// TwinCAT 3 PLC project EngineeringToolbox
// Title: EngineeringToolbox
// Company: Beckhoff Electronics Mfg
// Author: Daniel Schlingmann
// ProjectVersion: 3.1.2.3
// Description: Engineering Toolbox Library The library is provided "as-is" for TwinCAT3.1 by the Beckhoff Industry Management for Electronics Manufacturing. Please check the function "DisclaimerStatement : WSTRING[1500]" in additon to the following disclaimer: THE SOFTWARE IS PROVIDED "AS IS", WITHOUT WARRANTY OF ANY KIND, EXPRESS OR IMPLIED, INCLUDING BUT NOT LIMITED TO THE WARRANTIES OF MERCHANTABILITY, FITNESS FOR A PARTICULAR PURPOSE AND NONINFRINGEMENT. IN NO EVENT SHALL THE AUTHORS OR COPYRIGHT HOLDERS BE LIABLE FOR ANY CLAIM, DAMAGES OR OTHER LIABILITY, WHETHER IN AN ACTION OF CONTRACT, TORT OR OTHERWISE, ARISING FROM, OUT OF OR IN CONNECTION WITH THE SOFTWARE OR THE USE OR OTHER DEALINGS IN THE SOFTWARE.
// ProgramVersion: 3.1.4022.7
// libraries:
//   Tc2_Drive, * (Beckhoff Automation GmbH)
//   Tc2_EtherCAT, * (Beckhoff Automation GmbH)
//   Tc2_IoFunctions, * (Beckhoff Automation GmbH)
//   Tc2_Math, * (Beckhoff Automation GmbH)
//   Tc2_MC2, * (Beckhoff Automation GmbH)
//   Tc2_MC2_Camming, * (Beckhoff Automation GmbH)
//   Tc2_MC2_Drive, * (Beckhoff Automation GmbH)
//   Tc2_MC2_FlyingSaw, * (Beckhoff Automation GmbH)
//   Tc2_MDP, * (Beckhoff Automation GmbH)
//   Tc2_ModbusRTU, * (Beckhoff Automation GmbH)
//   Tc2_ModbusSrv, * (Beckhoff Automation GmbH)
//   Tc2_NC, * (Beckhoff Automation GmbH)
//   Tc2_NCI, * (Beckhoff Automation GmbH)
//   Tc2_NcKinematicTransformation, * (Beckhoff Automation GmbH)
//   Tc2_PlcInterpolation, * (Beckhoff Automation GmbH)
//   Tc2_SerialCom, * (Beckhoff Automation GmbH)
//   Tc2_Smtp, * (Beckhoff Automation GmbH)
//   Tc2_Standard, * (Beckhoff Automation GmbH)
//   Tc2_SUPS, * (Beckhoff Automation GmbH)
//   Tc2_System, * (Beckhoff Automation GmbH)
//   Tc2_TcpIp, * (Beckhoff Automation GmbH)
//   Tc2_Utilities, * (Beckhoff Automation GmbH)
//   Tc2_XmlDataSrv, * (Beckhoff Automation GmbH)
//   Tc3_Module, * (Beckhoff Automation GmbH)
//   Tc2_BackupRestoreEL6900,newest,Beckhoff Automation GmbH
// project tree:
//   GVLs/ Gvl.TcGVL, PARAM.TcGVL
//   POUs/BoundsCheck/ boundsError.TcPOU (not stored), boundsOK.TcPOU (not stored), checkBounds.TcPOU, CheckBoundsInfo.TcPOU
//   POUs/Connectivity/ADS/ AdsDataExchange.TcPOU (not stored)
//   POUs/Connectivity/ Ipv4Addr_TO_UDINT.TcPOU (not stored), U_DEVICE_COM_CACHE.TcDUT (not stored), U_IPv4Addr.TcDUT (not stored), isValidIPv4Addr.TcPOU
//   POUs/Connectivity/TF6310-TcpServer/DeviceCom/ TCPDeviceCom_SendRecBytes.TcPOU (not stored), TCPDeviceCom_SendRecString.TcPOU
//   POUs/Connectivity/TF6340-SerialCom/ComPortDeviceCom/ ComPortDeviceCom_BufferHandle.TcPOU, ComPortDeviceCom_SendRecBytes.TcPOU, ComPortDeviceCom_SendRecString.TcPOU (not stored), ComPortEL6x22BEasyConnect.TcPOU (not stored)
//   POUs/Connectivity/TF6340-SerialCom/ComPortBasic/ ComPortBackground.TcPOU (not stored), ComPortSendRec.TcPOU
//   POUs/Connectivity/TF625x-Modbus/Master/TF6250-ModbusTcpServer/TCP/ ModbusTcpMaster.TcPOU
//   POUs/Connectivity/TF625x-Modbus/Master/TF6250-ModbusTcpServer/UDP/ ModbusUdpMaster.TcPOU
//   POUs/Connectivity/TF625x-Modbus/Master/TF6255-ModbusRtu/ ModbusRtuMaster22B.TcPOU, ModbusRtuMaster5B.TcPOU (not stored), ModbusRtuMasterPC.TcPOU
//   POUs/Connectivity/TF625x-Modbus/Master/_Components/ ModbusJob.TcPOU (not stored), ModbusSlaveCom.TcPOU
//   POUs/Connectivity/TF625x-Modbus/Slave/ ModbusSlaveBase.TcPOU (not stored)
//   POUs/Connectivity/TF6310-TcpServer/TcpBasic/ TCPSendRecCtrl.TcPOU (not stored), TCPConnectionCtrl.TcPOU, TCPSocketCtrl.TcPOU (not stored)
//   POUs/Connectivity/TF6310-TcpServer/UdpBasic/ UDPSendRecCtrl.TcPOU (not stored), UDPServerCtrl.TcPOU (not stored), UDPSocketCtrl.TcPOU (not stored)
//   POUs/ControllerTools/ AverageFilter.TcPOU (not stored), PIDController.TcPOU (not stored), PT1Filter.TcPOU (not stored), signum.TcPOU (not stored), SlewRateLimitter.TcPOU, SlidingAverageExt.TcPOU, SlidingAverage.TcPOU, ThreePointController.TcPOU
//   POUs/DataBuffer/ DoubleBuffer.TcPOU (not stored), Quicksort.TcPOU (not stored)
//   POUs/DataBuffer/Fifo/ Fifo.TcPOU (not stored), FifoExt.TcPOU, FifoLRealSimple.TcPOU, FifoBase.TcPOU
//   POUs/DataBuffer/Ringbuffer/ RingbufferBase.TcPOU, Ringbuffer.TcPOU (not stored), RingbufferCharSimple.TcPOU (not stored), RingbufferExt.TcPOU (not stored), RingbufferByteSimple.TcPOU (not stored), RingbufferLRealSimple.TcPOU
//   POUs/EventLogger/ EventsWriteToLogbook.TcPOU (not stored), EVENT_HANDLING_CONFIG.TcDUT (not stored), getEventClassPriority.TcPOU (not stored), getEventClassText.TcPOU (not stored), SOURCE_ID.TcDUT (not stored)
//   POUs/EventLogger/ReadEvents/ EventlogRead.TcPOU (not stored), EVENTLOG_READ_DATA.TcDUT (not stored), EVENTLOG_READ_HANDLEINFO.TcDUT (not stored), EVENTLOG_READ_STREAM.TcDUT (not stored), EVENTLOG_READ_STREAM_DATA_RAW.TcDUT (not stored), EVENTLOG_READ_STREAM_DATA_RAW_EX.TcDUT
//   POUs/EventLogger/TriggerEvents/ EventHandling.TcPOU, EventHandlingGrp10.TcPOU (not stored), EventHandlingGrp25.TcPOU, EventHandlingGrp50.TcPOU (not stored), EventHandlingGrpCustomized.TcPOU (not stored), EventHandlingConfirmIsReq.TcPOU (not stored), EventHandlingStatisticInfo.TcPOU
//   POUs/Fieldbus/CANopen/ CANopenMasterDiag.TcPOU (not stored), CANopenMasterIO.TcPOU
//   POUs/Fieldbus/EAP/ EAP_PUB_SUB_IO.TcPOU (not stored), EAP_DEVICE_IO.TcPOU (not stored), EAP_PUB_VAR.TcPOU, EAP_SUB_VAR.TcPOU (not stored)
//   POUs/Fieldbus/EtherCAT/ EcCoEReadNewestDiagMsg.TcPOU, EcDiagBase.TcPOU, EcDiagBase_wEvents.TcPOU
//   POUs/Fieldbus/EtherCAT/_Components/ EcMasterIO.TcPOU (not stored), EcMasterSupervisor.TcPOU (not stored), EcSlavesDiag.TcPOU (not stored), EcSlaveSupervisor.TcPOU, EC_MASTER_DEVICE_STATE.TcDUT, EC_SLAVE_DIAG_INFO_DATA.TcDUT (not stored)
//   POUs/Fieldbus/Profibus/ ProfibusMasterDiag.TcPOU (not stored), ProfibusMasterIO.TcPOU (not stored)
//   POUs/Fieldbus/Profinet/ ProfinetControllerIO.TcPOU (not stored), ProfinetControllerIO_wEvents.TcPOU (not stored), ProfinetDeviceIO.TcPOU (not stored)
//   POUs/FileHandling/Basic/ FileHandling.TcPOU, ReadDirSimple.TcPOU (not stored), ReadDirSimpleExt.TcPOU
//   POUs/FileHandling/TF6421-XmlServer/ XmlReadWrite.TcPOU (not stored), XmlReadWriteWithBackupFile.TcPOU (not stored)
//   POUs/IO/Analog/ AnalogIn.TcPOU, AnalogIn32.TcPOU, AnalogInELMBase.TcPOU (not stored), AnalogInELMSingleSampleDINT.TcPOU, AnalogInELMSingleSampleREAL.TcPOU (not stored), AnalogInREAL.TcPOU, AnalogOut.TcPOU (not stored)
//   POUs/IO/ BlowOffSensors.TcPOU (not stored), Button.TcPOU, ButtonExt.TcPOU (not stored), Fuse.TcPOU (not stored), InOut.TcPOU (not stored), InOutExt.TcPOU (not stored), Input.TcPOU (not stored), Output.TcPOU (not stored)
//   POUs/IO/Cylinder/ Cylinder.TcPOU, CylinderExt.TcPOU (not stored), CylinderType4.TcPOU, I_Cylinder.TcIO (not stored)
//   POUs/IO/Drives/ AxDriveBase.TcPOU (not stored), AxDriveGetRef.TcPOU (not stored), I_AxDriveBase.TcIO
//   POUs/IO/Drives/CoE/ AxDriveCoE.TcPOU, AxDriveCoE_wEvents.TcPOU, CiA_DS402Controlword.TcPOU (not stored), CiA_DS402Statusword.TcPOU (not stored), eCiA_DS402_CONTROL_CMD.TcDUT, eCiA_DS402_STATUS_STATE.TcDUT (not stored)
//   POUs/IO/Drives/CoE/EL72xx/ AxDriveCoE_EL72xxParam.TcPOU (not stored), CiA_DS402StatuswordEx7xxx.TcPOU
//   POUs/IO/Drives/DC/Ey73xx/ AxDriveDC.TcPOU (not stored), AxDriveDC_wEvents.TcPOU (not stored)
//   POUs/IO/Drives/SoE/ AxDriveSoE_Ax5000CommutationCalib.TcPOU (not stored), AxDriveSoE_Ax5000CalcPower.TcPOU (not stored), AxDriveSoE_Ax5000SwitchParamSet.TcPOU (not stored), Ax580x.TcPOU (not stored), AxDriveSoE_Ax5000.TcPOU, AxDriveSoE_Ax5000Param.TcPOU, AxDriveSoE_Ax5000wEvents.TcPOU, AxDriveSoE_Rexroth.TcPOU (not stored)
//   POUs/IO/Drives/SoE/Ax5000ParamSTRUCTs/P/ AX5000_P_0001.TcDUT (not stored), AX5000_P_0002.TcDUT (not stored), AX5000_P_0003.TcDUT (not stored), AX5000_P_0004.TcDUT (not stored), AX5000_P_0009.TcDUT, AX5000_P_0010.TcDUT, AX5000_P_0020.TcDUT, AX5000_P_0021.TcDUT (not stored), AX5000_P_0040.TcDUT (not stored), AX5000_P_0050.TcDUT, AX5000_P_0051.TcDUT, AX5000_P_0052.TcDUT (not stored), AX5000_P_0053.TcDUT, AX5000_P_0054.TcDUT (not stored), AX5000_P_0055.TcDUT (not stored), AX5000_P_0056.TcDUT, AX5000_P_0057.TcDUT, AX5000_P_0058.TcDUT (not stored), AX5000_P_0059.TcDUT, AX5000_P_0060.TcDUT (not stored), AX5000_P_0061.TcDUT, AX5000_P_0062.TcDUT (not stored), AX5000_P_0063.TcDUT (not stored), AX5000_P_0064.TcDUT (not stored), AX5000_P_0065.TcDUT, AX5000_P_0066.TcDUT (not stored), AX5000_P_0067.TcDUT, AX5000_P_0068.TcDUT (not stored), AX5000_P_0069.TcDUT (not stored), AX5000_P_0070.TcDUT, AX5000_P_0071.TcDUT (not stored), AX5000_P_0072.TcDUT (not stored), AX5000_P_0073.TcDUT (not stored), AX5000_P_0074.TcDUT (not stored), AX5000_P_0075.TcDUT (not stored), AX5000_P_0076.TcDUT (not stored), AX5000_P_0077.TcDUT (not stored), AX5000_P_0078.TcDUT, AX5000_P_0088.TcDUT, AX5000_P_0089.TcDUT (not stored), AX5000_P_0090.TcDUT (not stored), AX5000_P_0091.TcDUT (not stored), AX5000_P_0092.TcDUT (not stored), AX5000_P_0093.TcDUT, AX5000_P_0096.TcDUT (not stored), AX5000_P_0097.TcDUT, AX5000_P_0098_beckhoff.TcDUT (not stored), AX5000_P_0098_beckhoff_electrical_data.TcDUT (not stored), AX5000_P_0099.TcDUT (not stored), AX5000_P_0100.TcDUT (not stored), AX5000_P_0101.TcDUT (not stored), AX5000_P_0102.TcDUT (not stored), AX5000_P_0103.TcDUT (not stored), AX5000_P_0104.TcDUT (not stored), AX5000_P_0105.TcDUT (not stored), AX5000_P_0106.TcDUT (not stored), AX5000_P_0107.TcDUT (not stored), AX5000_P_0108.TcDUT (not stored), AX5000_P_0109.TcDUT (not stored), AX5000_P_0110.TcDUT, AX5000_P_0111.TcDUT (not stored), AX5000_P_0112.TcDUT (not stored), AX5000_P_0113.TcDUT (not stored), AX5000_P_0114.TcDUT, AX5000_P_0115.TcDUT (not stored), AX5000_P_0116.TcDUT (not stored), AX5000_P_0117.TcDUT (not stored), AX5000_P_0118.TcDUT (not stored), AX5000_P_0119.TcDUT, AX5000_P_0125.TcDUT (not stored), AX5000_P_0126.TcDUT (not stored), AX5000_P_0127.TcDUT (not stored), AX5000_P_0128.TcDUT (not stored), AX5000_P_0150.TcDUT (not stored), AX5000_P_0151.TcDUT (not stored), AX5000_P_0152.TcDUT, AX5000_P_0153.TcDUT (not stored), AX5000_P_0154.TcDUT, AX5000_P_0155.TcDUT (not stored), AX5000_P_0158.TcDUT, AX5000_P_0159.TcDUT, AX5000_P_0160.TcDUT (not stored), AX5000_P_0161.TcDUT (not stored), AX5000_P_0162.TcDUT, AX5000_P_0163.TcDUT (not stored), AX5000_P_0165.TcDUT (not stored), AX5000_P_0166.TcDUT, AX5000_P_0167.TcDUT (not stored), AX5000_P_0168.TcDUT (not stored), AX5000_P_0169.TcDUT, AX5000_P_0170.TcDUT (not stored), AX5000_P_0171.TcDUT (not stored), AX5000_P_0180.TcDUT (not stored), AX5000_P_0181.TcDUT (not stored), AX5000_P_0182.TcDUT (not stored), AX5000_P_0183.TcDUT (not stored), AX5000_P_0184.TcDUT (not stored), AX5000_P_0185.TcDUT (not stored), AX5000_P_0188.TcDUT, AX5000_P_0189.TcDUT (not stored), AX5000_P_0192.TcDUT (not stored), AX5000_P_0193.TcDUT (not stored), AX5000_P_0196.TcDUT, AX5000_P_0198.TcDUT (not stored), AX5000_P_0199.TcDUT (not stored), AX5000_P_0200.TcDUT (not stored), AX5000_P_0201.TcDUT (not stored), AX5000_P_0202.TcDUT (not stored), AX5000_P_0203.TcDUT (not stored), AX5000_P_0204.TcDUT (not stored), AX5000_P_0205.TcDUT, AX5000_P_0206.TcDUT (not stored), AX5000_P_0207.TcDUT, AX5000_P_0208.TcDUT, AX5000_P_0209.TcDUT (not stored), AX5000_P_0210.TcDUT (not stored), AX5000_P_0211.TcDUT (not stored), AX5000_P_0212.TcDUT, AX5000_P_0213.TcDUT, AX5000_P_0214.TcDUT (not stored), AX5000_P_0215.TcDUT, AX5000_P_0216.TcDUT (not stored), AX5000_P_0217.TcDUT (not stored), AX5000_P_0218.TcDUT (not stored), AX5000_P_0219.TcDUT, AX5000_P_0220.TcDUT (not stored), AX5000_P_0221.TcDUT (not stored), AX5000_P_0250.TcDUT (not stored), AX5000_P_0251.TcDUT, AX5000_P_0252.TcDUT, AX5000_P_0253.TcDUT, AX5000_P_0254.TcDUT (not stored), AX5000_P_0255.TcDUT, AX5000_P_0256.TcDUT, AX5000_P_0270.TcDUT (not stored), AX5000_P_0271.TcDUT (not stored), AX5000_P_0272.TcDUT (not stored), AX5000_P_0273.TcDUT, AX5000_P_0274.TcDUT (not stored), AX5000_P_0275.TcDUT, AX5000_P_0276.TcDUT (not stored), AX5000_P_0277.TcDUT (not stored), AX5000_P_0278.TcDUT (not stored), AX5000_P_0300.TcDUT (not stored), AX5000_P_0301.TcDUT, AX5000_P_0302.TcDUT (not stored), AX5000_P_0303.TcDUT (not stored), AX5000_P_0304.TcDUT, AX5000_P_0305.TcDUT (not stored), AX5000_P_0306.TcDUT (not stored), AX5000_P_0307.TcDUT (not stored), AX5000_P_0308.TcDUT, AX5000_P_0309.TcDUT (not stored), AX5000_P_0310.TcDUT, AX5000_P_0311.TcDUT (not stored), AX5000_P_0312.TcDUT, AX5000_P_0313.TcDUT (not stored), AX5000_P_0314.TcDUT, AX5000_P_0315.TcDUT, AX5000_P_0316.TcDUT, AX5000_P_0317.TcDUT (not stored), AX5000_P_0320.TcDUT (not stored), AX5000_P_0321.TcDUT (not stored), AX5000_P_0322.TcDUT (not stored), AX5000_P_0323.TcDUT, AX5000_P_0324.TcDUT (not stored), AX5000_P_0325.TcDUT (not stored), AX5000_P_0326.TcDUT (not stored), AX5000_P_0350.TcDUT, AX5000_P_0351.TcDUT (not stored), AX5000_P_0352.TcDUT (not stored), AX5000_P_0353.TcDUT (not stored), AX5000_P_0354.TcDUT (not stored), AX5000_P_0356.TcDUT, AX5000_P_0360.TcDUT, AX5000_P_0361.TcDUT (not stored), AX5000_P_0400.TcDUT (not stored), AX5000_P_0401.TcDUT (not stored), AX5000_P_0402.TcDUT, AX5000_P_0451.TcDUT, AX5000_P_0452.TcDUT (not stored), AX5000_P_0453.TcDUT (not stored), AX5000_P_0454.TcDUT (not stored), AX5000_P_0455.TcDUT (not stored), AX5000_P_0456.TcDUT (not stored), AX5000_P_0457.TcDUT, AX5000_P_0458.TcDUT (not stored), AX5000_P_0459.TcDUT, AX5000_P_0460.TcDUT (not stored), AX5000_P_0461.TcDUT, AX5000_P_0462.TcDUT (not stored), AX5000_P_0463.TcDUT (not stored), AX5000_P_0464.TcDUT (not stored), AX5000_P_0502.TcDUT (not stored), AX5000_P_0503.TcDUT (not stored), AX5000_P_0504.TcDUT, AX5000_P_0505.TcDUT (not stored), AX5000_P_0511.TcDUT, AX5000_P_0512.TcDUT (not stored), AX5000_P_0513.TcDUT (not stored), AX5000_P_0514.TcDUT (not stored), AX5000_P_0515.TcDUT, AX5000_P_0516.TcDUT (not stored), AX5000_P_0517.TcDUT, AX5000_P_0518.TcDUT, AX5000_P_0552.TcDUT (not stored), AX5000_P_0553.TcDUT, AX5000_P_0554.TcDUT, AX5000_P_0555.TcDUT (not stored), AX5000_P_0556.TcDUT (not stored), AX5000_P_0557.TcDUT (not stored), AX5000_P_0558.TcDUT (not stored), AX5000_P_0601.TcDUT, AX5000_P_0602.TcDUT (not stored), AX5000_P_0610.TcDUT (not stored), AX5000_P_0611.TcDUT (not stored), AX5000_P_0800.TcDUT (not stored), AX5000_P_0801.TcDUT, AX5000_P_0802.TcDUT (not stored), AX5000_P_0804.TcDUT (not stored), AX5000_P_0805.TcDUT (not stored), AX5000_P_0806.TcDUT, AX5000_P_0810.TcDUT (not stored), AX5000_P_0811.TcDUT (not stored), AX5000_P_0850.TcDUT, AX5000_P_0851.TcDUT, AX5000_P_0900.TcDUT (not stored), AX5000_P_0901.TcDUT (not stored), AX5000_P_0902.TcDUT, AX5000_P_0904.TcDUT (not stored), AX5000_P_0905.TcDUT (not stored), AX5000_P_0906.TcDUT (not stored), AX5000_P_0912.TcDUT, AX5000_P_1000.TcDUT (not stored), AX5000_P_1001.TcDUT, AX5000_P_1002.TcDUT (not stored), AX5000_P_1003.TcDUT (not stored), AX5000_P_1004.TcDUT (not stored), AX5000_P_1005.TcDUT (not stored), AX5000_P_1006.TcDUT (not stored), AX5000_P_1007.TcDUT, AX5000_P_1008.TcDUT, AX5000_P_1009.TcDUT (not stored), AX5000_P_1010.TcDUT (not stored), AX5000_P_1011.TcDUT (not stored), AX5000_P_1012.TcDUT (not stored), AX5000_P_1020.TcDUT (not stored), AX5000_P_1021.TcDUT (not stored), AX5000_P_1022.TcDUT, AX5000_P_2000.TcDUT, AX5000_P_2001.TcDUT, AX5000_P_2002.TcDUT
//   POUs/IO/Drives/SoE/Ax5000ParamSTRUCTs/S/ AX5000_S_0001.TcDUT, AX5000_S_0002.TcDUT (not stored), AX5000_S_0007.TcDUT (not stored), AX5000_S_0011.TcDUT, AX5000_S_0012.TcDUT (not stored), AX5000_S_0013.TcDUT, AX5000_S_0015.TcDUT, AX5000_S_0016.TcDUT (not stored), AX5000_S_0017.TcDUT (not stored), AX5000_S_0018.TcDUT, AX5000_S_0024.TcDUT (not stored), AX5000_S_0029.TcDUT (not stored), AX5000_S_0030.TcDUT, AX5000_S_0031.TcDUT, AX5000_S_0032.TcDUT (not stored), AX5000_S_0033.TcDUT (not stored), AX5000_S_0034.TcDUT (not stored), AX5000_S_0035.TcDUT (not stored), AX5000_S_0036.TcDUT (not stored), AX5000_S_0037.TcDUT, AX5000_S_0040.TcDUT (not stored), AX5000_S_0043.TcDUT (not stored), AX5000_S_0044.TcDUT (not stored), AX5000_S_0045.TcDUT (not stored), AX5000_S_0046.TcDUT (not stored), AX5000_S_0047.TcDUT (not stored), AX5000_S_0048.TcDUT, AX5000_S_0051.TcDUT (not stored), AX5000_S_0053.TcDUT, AX5000_S_0055.TcDUT (not stored), AX5000_S_0076.TcDUT (not stored), AX5000_S_0079.TcDUT (not stored), AX5000_S_0080.TcDUT, AX5000_S_0081.TcDUT, AX5000_S_0082.TcDUT (not stored), AX5000_S_0083.TcDUT (not stored), AX5000_S_0084.TcDUT (not stored), AX5000_S_0085.TcDUT (not stored), AX5000_S_0086.TcDUT, AX5000_S_0091.TcDUT, AX5000_S_0092.TcDUT (not stored), AX5000_S_0095.TcDUT, AX5000_S_0099.TcDUT, AX5000_S_0100.TcDUT, AX5000_S_0101.TcDUT (not stored), AX5000_S_0103.TcDUT (not stored), AX5000_S_0104.TcDUT, AX5000_S_0106.TcDUT, AX5000_S_0107.TcDUT (not stored), AX5000_S_0109.TcDUT (not stored), AX5000_S_0110.TcDUT (not stored), AX5000_S_0111.TcDUT, AX5000_S_0112.TcDUT (not stored), AX5000_S_0113.TcDUT (not stored), AX5000_S_0119.TcDUT, AX5000_S_0120.TcDUT (not stored), AX5000_S_0124.TcDUT (not stored), AX5000_S_0126.TcDUT, AX5000_S_0130.TcDUT (not stored), AX5000_S_0131.TcDUT, AX5000_S_0134.TcDUT, AX5000_S_0135.TcDUT (not stored), AX5000_S_0136.TcDUT (not stored), AX5000_S_0137.TcDUT (not stored), AX5000_S_0143.TcDUT (not stored), AX5000_S_0149.TcDUT (not stored), AX5000_S_0159.TcDUT, AX5000_S_0160.TcDUT, AX5000_S_0161.TcDUT, AX5000_S_0162.TcDUT, AX5000_S_0163.TcDUT, AX5000_S_0169.TcDUT (not stored), AX5000_S_0170.TcDUT (not stored), AX5000_S_0179.TcDUT, AX5000_S_0185.TcDUT, AX5000_S_0186.TcDUT (not stored), AX5000_S_0187.TcDUT, AX5000_S_0188.TcDUT, AX5000_S_0189.TcDUT (not stored), AX5000_S_0196.TcDUT (not stored), AX5000_S_0200.TcDUT, AX5000_S_0201.TcDUT (not stored), AX5000_S_0203.TcDUT (not stored), AX5000_S_0204.TcDUT (not stored), AX5000_S_0206.TcDUT (not stored), AX5000_S_0207.TcDUT (not stored), AX5000_S_0216.TcDUT, AX5000_S_0217.TcDUT, AX5000_S_0219.TcDUT (not stored), AX5000_S_0254.TcDUT (not stored), AX5000_S_0256.TcDUT (not stored), AX5000_S_0257.TcDUT (not stored), AX5000_S_0267.TcDUT, AX5000_S_0273.TcDUT (not stored), AX5000_S_0274.TcDUT, AX5000_S_0292.TcDUT (not stored), AX5000_S_0295.TcDUT (not stored), AX5000_S_0296.TcDUT (not stored), AX5000_S_0347.TcDUT (not stored), AX5000_S_0348.TcDUT (not stored), AX5000_S_0372.TcDUT, AX5000_S_0374.TcDUT (not stored), AX5000_S_0375.TcDUT, AX5000_S_0380.TcDUT, AX5000_S_0381.TcDUT (not stored), AX5000_S_0383.TcDUT, AX5000_S_0384.TcDUT (not stored), AX5000_S_0390.TcDUT (not stored), AX5000_S_0403.TcDUT (not stored), AX5000_S_0405.TcDUT (not stored), AX5000_S_0409.TcDUT (not stored), AX5000_S_0410.TcDUT (not stored), AX5000_S_0429.TcDUT, AX5000_S_0432.TcDUT (not stored), AX5000_S_0435.TcDUT, AX5000_S_0436.TcDUT (not stored)
//   POUs/IO/Drives/Stepper/ AxDriveStepper.TcPOU, AxDriveStepperParam.TcPOU (not stored), AxDriveStepper_wEvents.TcPOU (not stored)
//   POUs/IO/EL-EP/ AnalogOut_EL2535.TcPOU (not stored), EL1262_Base.TcPOU (not stored), EL3681.TcPOU (not stored), EL1904.TcPOU (not stored), EL69xx.TcPOU, EL3356.TcPOU (not stored), Eyx9xx.TcPOU, ZB8610.TcPOU
//   POUs/IO/EL-EP/EL9x/ EL9501.TcPOU (not stored), EL9576.TcPOU (not stored), EL95xxPowerTerminal.TcPOU, ELSystemTerminal.TcPOU
//   POUs/IO/_EcSlaveFWUpdater/ EcSlaveDevFWUpdater.TcPOU (not stored)
//   POUs/IO/_EcSlaveInfoDataIO/ EcSlaveInfoData.TcPOU (not stored), EcSlaveInfoDataExt.TcPOU (not stored), I_EcSlaveInfoData.TcIO
//   POUs/IO/EL-EP/EL3403/ EL3403.TcPOU (not stored), EL3403Logic.TcPOU
//   POUs/IO/EL-EP/EP92xxPwrBox/ EP9214.TcPOU, EP9214_CHANNEL.TcPOU (not stored), EP9224_0037.TcPOU, EP9224_0037_CHANNEL.TcPOU
//   POUs/IO/FreqConv/EtherCAT/DS402/ EcFcDS402_ComBase.TcPOU (not stored)
//   POUs/IO/FreqConv/ IOFcCom.TcPOU
//   POUs/IO/Motors/ IOMotor.TcPOU (not stored), IOMotor2Dir.TcPOU (not stored), IOMotorStarDelta.TcPOU (not stored)
//   POUs/IO/[underDev]/ Cylinder_wUnitItf.TcPOU
//   POUs/IO/_ItfActuators/ I_ActuatorBase.TcIO (not stored), I_ActuatorEnableDisable.TcIO (not stored), I_ActuatorFwdRev.TcIO, I_ActuatorFwdBwd.TcIO, I_ActuatorLeftRight.TcIO, I_ActuatorOnOff.TcIO (not stored), I_ActuatorOpenClose.TcIO (not stored), I_ActuatorPosNeg.TcIO (not stored), I_ActuatorStartStop.TcIO (not stored), I_ActuatorUpDown.TcIO (not stored), I_ActuatorWorkBase.TcIO (not stored)
//   POUs/IpcDiag/MDP/InfoModuls/ MDP_CPU.TcPOU, MDP_Fan.TcPOU, MDP_Mainboard.TcPOU (not stored), MDP_RaidSimple.TcPOU (not stored), MDP_ReadModulList.TcPOU (not stored), MDP_SiliconDrives.TcPOU, MDP_UPS.TcPOU (not stored)
//   POUs/IpcDiag/MDP/ MDP_Info.TcPOU, MDP_IpcDiag.TcPOU (not stored), MDP_IpcDiag_wEvents.TcPOU (not stored)
//   POUs/IpcDiag/ UPSStatus.TcPOU (not stored)
//   POUs/Logging/ DataFileLogger.TcPOU, DataUdpLogger.TcPOU (not stored), I_LogbookSubscriber.TcIO (not stored), I_Logbook.TcIO (not stored), Logbook.TcPOU (not stored), LogbookData.TcDUT, LogbookPuplisher.TcPOU, LogbookSubEventLog.TcPOU (not stored), LogbookSubSendMail.TcPOU, adsLogError.TcPOU, adsLogHint.TcPOU (not stored), adsLogWarn.TcPOU, LogbookSubSysLog.TcPOU, LogbookSubWriteFile.TcPOU, Logbook_wEventClass.TcPOU, adsLogwTcEventClass.TcPOU (not stored)
//   POUs/Motion/TF50xx-NC/00_Base/ I_AxNcPTP.TcIO (not stored), AxFbBase.TcPOU, AxRWParaBase.TcPOU (not stored), I_AxNcBase.TcIO
//   POUs/Motion/TF50xx-NC/02_Options/Parameter/ AxPara.TcPOU (not stored), AxParaCtrl.TcPOU
//   POUs/Motion/TF50xx-NC/03_Utilities/ AxAutoWriteSoftLimit.TcPOU, CoordinateTransformation2D.TcPOU (not stored), AxCalcPosBias.TcPOU, AxResonanceAvoidance.TcPOU (excluded from build), AxSoftSyncDistance.TcPOU (not stored), AxStatemodel.TcPOU (not stored), AxAutoFct.TcPOU (not stored), AX_JOB.TcPOU (not stored), getOvrVelo.TcPOU
//   POUs/Motion/TF50xx-NC/ AxNcPTPwJobs.TcPOU (not stored), AxNcBaseExt.TcPOU (not stored), AxNcPtpGear.TcPOU, AxNcBase.TcPOU, AxNcPTP.TcPOU (not stored)
//   POUs/Motion/TF5100-NCI/ NciChannel_wEvents.TcPOU (not stored), NciChannel.TcPOU (not stored)
//   POUs/Motion/TF511x-KIN/03_DUTs/Positions/ KIN_POSITIONS.TcPOU (not stored), KIN_POSITIONS_ACS_DUT.TcDUT (not stored), KIN_POSITIONS_MCS_DUT.TcDUT, U_KIN_POSITIONS.TcDUT
//   POUs/Motion/TF511x-KIN/03_DUTs/Trafo/ KIN_CALCTRAFO_AXPOS_PARAM.TcPOU (not stored), KIN_STATE_OBSERVER_OID_PARAM.TcPOU (not stored), KIN_STATICTRAFO_PARAM.TcPOU (not stored), KIN_TOOLTRAFO_PARAM.TcPOU, UCS.TcPOU (not stored)
//   POUs/Motion/ VALUE_3D.TcPOU (not stored), VALUE_3D_DUT.TcDUT (not stored), VALUE_6D.TcPOU (not stored), VALUE_6D_DUT.TcDUT
//   POUs/Safety/Diag/ SafetyLogicAndIOTerminalDiag.TcPOU (not stored), SafetyIODeviceDiagRead.TcPOU (not stored), SafetyIODeviceDiag_wEvents.TcPOU, SafetyIOsDiag.TcPOU, SafetyLogicTerminalDiag.TcPOU, SafetyPlcTerminalDiag.TcPOU
//   POUs/StringHelper/ CHR_TO_STR.TcPOU, cutStrNumberToSeperator.TcPOU (not stored), cutStrToSeperator2.TcPOU, replaceUmlauts.TcPOU, stringCmp.TcPOU, STR_TO_ASC.TcPOU (not stored), cutStrToSeperator.TcPOU (not stored), cutWStrToSeperator.TcPOU (not stored), DWORD_TO_BINSTR_EXT.TcPOU (not stored), DWORD_TO_HEXSTR_EXT.TcPOU (not stored), getCntCharInStr.TcPOU (not stored), getCntCharInWStr.TcPOU, isWStringNumeric.TcPOU (not stored), HEXSTR_TO_DWORD.TcPOU, HEXSTR_TO_LWORD.TcPOU, INSERT_EXT.TcPOU, LWORD_TO_BINSTR_EXT.TcPOU, LWORD_TO_HEXSTR_EXT.TcPOU, readStrToSeperator.TcPOU, replaceInString.TcPOU (not stored), getFilledString.TcPOU (not stored), isStringNumeric.TcPOU (not stored), readWStrToSeperator.TcPOU (not stored), replaceInWString.TcPOU, U_MAX_STRING.TcDUT, U_MAX_WSTRING.TcDUT, WINSERT_EXT.TcPOU (not stored)
//   POUs/System/ SystemInfo.TcPOU (not stored), SystemInfo64.TcPOU (not stored) (excluded from build), SystemPulses.TcPOU (not stored), TaskInfo.TcPOU (not stored)
//   POUs/TimeHelper/ PartsPerTime.TcPOU (not stored), createTOD.TcPOU (not stored), getDateAndTimeDelta.TcPOU (not stored), getTonCountdown.TcPOU, LivebitCheck.TcPOU (not stored), Ontime.TcPOU (not stored), OntimeExt.TcPOU, OntimeSimple.TcPOU (not stored), Pulse.TcPOU (not stored), SensorTimeoutCheck.TcPOU, systemtimeInCam.TcPOU (not stored), systemtimeCmp.TcPOU (not stored), systemtimeInWin.TcPOU, TimeSwitch.TcPOU (not stored), TONRecord.TcPOU (not stored), TONTOF.TcPOU (not stored), VeloLinearMeasurement.TcPOU
//   POUs/_Miscellaneous/64BitFunctions/ CLEARBIT64.TcPOU (not stored), CSETBIT64.TcPOU, GETBIT64.TcPOU, SETBIT64.TcPOU
//   POUs/_Miscellaneous/Conversions/ TO_FMREAL.TcPOU, ADSERROR_TO_HRESULT.TcPOU (not stored), DWORD_TO_REAL_EX.TcPOU (not stored), HRESULT_TO_ADSERROR.TcPOU, REAL_TO_FMLREAL.TcPOU, LWORD_TO_LREAL_EX.TcPOU (not stored), SWAP_BYTES_OF_WORDS.TcPOU (not stored), SWAP_WORDS_OF_DWORD.TcPOU (not stored), SWAP_WORDS_OF_LWORD.TcPOU (not stored), ADSERROR_TO_WIN32ERROR.TcPOU (not stored), ADSERROR_TO_WSERROR.TcPOU, C_TO_F.TcPOU (not stored), DEGREES_TO_RPM.TcPOU (not stored), F_TO_C.TcPOU (not stored), GF_TO_N.TcPOU (not stored), TO_FMLREAL.TcPOU (not stored), MMIN_TO_MMS.TcPOU (not stored), MMS_TO_MMIN.TcPOU (not stored), N_TO_GF.TcPOU (not stored), RPM_TO_DEGREES.TcPOU (not stored)
//   POUs/_Miscellaneous/ nextIdx.TcPOU (not stored), scale2.TcPOU (not stored), TC_VN_COLORS.TcDUT (not stored) (excluded from build), FbBase.TcPOU (not stored), CAM.TcPOU (not stored), CAM3D.TcPOU (not stored), COLOR.TcDUT (not stored), ERROR_HDL.TcPOU (not stored), FbBaseExt.TcPOU (not stored), FbBaseOutputs.TcPOU, getNoOfBits.TcPOU (not stored), LCID.TcDUT (not stored), eLCID.TcDUT (not stored), LOGx.TcPOU, OEECalculation.TcPOU (not stored), polynomial.TcPOU (not stored), RF_TRIG.TcPOU, scale.TcPOU, SEQUENCE_HDL.TcPOU, setNoOfBits.TcPOU (not stored), TEST_FB.TcPOU (not stored), TOGGLE.TcPOU (not stored), U_32BIT_DATATYPE.TcDUT, U_64BIT_DATATYPE.TcDUT, WIN.TcPOU (not stored)
//   POUs/Safety/ SafetyCircuit.TcPOU, SafetyGroupIO.TcPOU (not stored), SafetyPlcBackupRestore.TcPOU (not stored), SAFETY_CIRCUIT_STATUS.TcDUT (not stored)
//   POUs/Statemodel/control/ I_StatemodelBase.TcIO (not stored), I_Statemodel.TcIO (not stored), Statemodel.TcPOU
//   POUs/Statemodel/ eMODE.TcDUT (not stored), eSTATE.TcDUT
//   POUs/Statemodel/UnitTemplate/ I_Statemodel_Unit.TcIO, Statemodel_Unit.TcPOU
//   POUs/Motion/TF50xx-NC/01_Main/ AxAdmin.TcPOU, AxHoming.TcPOU (not stored), AxMotion.TcPOU
//   POUs/Motion/TF50xx-NC/02_Options/Motion/ AxSuperposition.TcPOU (not stored), AxMoveSinus.TcPOU (not stored), AxHomingOnBlock.TcPOU (not stored)
//   POUs/Motion/TF5100-NCI/01_Main/ NciAdmin.TcPOU (not stored), NciGrp.TcPOU (not stored), NciItp.TcPOU (not stored), NciMotion.TcPOU (not stored), NCI_REF.TcPOU
//   POUs/Motion/TF5100-NCI/02_Options/Error/ NciChnEventHandling.TcPOU (not stored), NciEventHandling.TcPOU (not stored)
//   POUs/Motion/TF5100-NCI/02_Options/MFunctions/ NciMFnc.TcPOU (not stored)
//   POUs/Motion/TF5100-NCI/02_Options/PlcItp/ NciCreateItpTable.TcPOU (not stored), NciCreateItpTableEntryTemplate.TcPOU (not stored)
//   POUs/Motion/TF5100-NCI/02_Options/RParameter/ NCiReadWriteRParam.TcPOU (not stored)
//   POUs/Motion/TF511x-KIN/01_Main/ KinAdmin.TcPOU, KIN_REF.TcPOU
//   POUs/Motion/TF511x-KIN/02_Options/ KinLockUnlockTrafoParam.TcPOU, KinWriteToolTrafoParam.TcPOU (not stored), KinWriteUCSTrafoParam.TcPOU (not stored)
//   POUs/Motion/TF511x-KIN/ KinChannel.TcPOU (not stored)
//   POUs/Motion/TF50xx-NC/02_Options/Coupling/ AxCamming.TcPOU (not stored), AxFlyingSaw.TcPOU, AxGear.TcPOU (not stored)
//   POUs/Motion/TF50xx-NC/02_Options/Error/ AxNcEventHandling.TcPOU, AxEventHandling.TcPOU (not stored)
//   POUs/Motion/TF50xx-NC/02_Options/Phasing/ AxPhasing.TcPOU (not stored)
//   POUs/Motion/TF50xx-NC/02_Options/TouchProbe/ AxTouchProbe.TcPOU (not stored)
//   POUs/StringHelper/ExtendedString/ ExtString.TcPOU (not stored), ExtWString.TcPOU (not stored), T_EXT_STRING.TcDUT, T_EXT_WSTRING.TcDUT
//   POUs/TimeHelper/Conversions/ FILETIME_TO_DATE.TcPOU, LREAL_TO_TIME_SEC.TcPOU, FILETIME_TO_TOD.TcPOU (not stored), SYSTEMTIME_TO_TIME.TcPOU (not stored), SYSTEMTIME_TO_TIME_EX.TcPOU (not stored), SYSTEMTIME_TO_TOD.TcPOU, SYSTEMTIME_TO_DATE.TcPOU, TIME_TO_FMRLREAL.TcPOU (not stored), TIME_TO_SYSTEMTIME.TcPOU (not stored)
//   Version/ disclaimerStatement.TcPOU, Global_Version.TcGVL

// ---- POUs/EventLogger/ReadEvents/EVENTLOG_READ_STREAM_DATA_RAW_EX.TcDUT
TYPE EVENTLOG_READ_STREAM_DATA_RAW_EX :
STRUCT
	cb				: WORD;			//Complete size OF the structure including data
	cbFmt			: WORD;			//Size OF the format STRING
	cbData			: WORD;			//Size OF the data
	Temp			: ARRAY [PARAM.EVENT_HANDLING_CONFIG.EVENTLOG_READ_MSG_LEN_MIN..PARAM.EVENT_HANDLING_CONFIG.EVENTLOG_READ_MSG_LEN_MAX] OF BYTE;
	
END_STRUCT
END_TYPE

// ---- POUs/Fieldbus/EtherCAT/_Components/EC_MASTER_DEVICE_STATE.TcDUT
TYPE EC_MASTER_DEVICE_STATE :
STRUCT
	NoError						: BOOL;//0x0000 = Link error 
	LinkError 					: BOOL;//0x0001 = Link error
	IOLockedAfterLinkError	    : BOOL;//0x0002 = I/O locked after link error (I/O reset required)
	LinkErrorRedMode			: BOOL;//0x0004 = Link error (redundancy adapter)
	MissingOneFrmInRedMode      : BOOL;//0x0008 = Missing one frame (redundancy mode)
	OutOfSendResources          : BOOL;//0x0010 = Out of send resources (I/O reset required)
	WatchdogTriggered 		    : BOOL;//0x0020 = Watchdog triggered
	EthernetDriverNotFound 	    : BOOL;//0x0040 = Ethernet driver (miniport) not found
	IOResetActive 			    : BOOL;//0x0080 = I/O reset active
	AtLeastOneSlaveInINIT       : BOOL;//0x0100 = At least one device in 'INIT' 
	AtLeastOneSlaveInPREOP      : BOOL;//0x0200 = At least one device in 'PRE-OP' 
	AtLeastOneSlaveInSAFEOP     : BOOL;//0x0400 = At least one device in 'SAFE-OP' 
	AtLeastOneSlaveInERROR     	: BOOL;//0x0800 = AT least one device indicates an error state 																	
	DcNotInSync 		        : BOOL;//0x1000 = DC NOT in sync
END_STRUCT
END_TYPE

// ---- POUs/IO/Drives/CoE/eCiA_DS402_CONTROL_CMD.TcDUT
{attribute 'qualified_only'}
{attribute 'to_string'}
TYPE eCiA_DS402_CONTROL_CMD :
(
	DISABLE_VOLTAGE											:= 2#0000_0000, //2#0xxx_xx0x -> back to switch on disabled
	SHUTDOWN												:= 2#0000_0110, //2#0xxx_x110 -> Voltage Enable - Ready to switch on
 	SWITCH_ON												:= 2#0000_0111, //2#0xxx_0111 -> Switched On = Disable operation (Switch on + NOT Enable operation)
	ENABLE_OPERATION										:= 2#0000_1111, //2#0xx0_1111 -> Operation enabled (Enable Voltage + Quick Stop OK + Switch on + Enable operation)	
	QUICK_STOP												:= 2#0000_1011, //2#0xxx_x01x 
	FAULT_RESET												:= 2#1000_0000  //2#1xxx_xxxx 
);
END_TYPE

// ---- POUs/IO/Drives/SoE/Ax5000ParamSTRUCTs/P/AX5000_P_0009.TcDUT
TYPE AX5000_P_0009 :
STRUCT
	Synchronisations_mode:UINT;
END_STRUCT
END_TYPE

// ---- POUs/IO/Drives/SoE/Ax5000ParamSTRUCTs/P/AX5000_P_0010.TcDUT
TYPE AX5000_P_0010 :
STRUCT
	Synchronization_mode:ARRAY[0..3] OF UINT;
END_STRUCT
END_TYPE

// ---- POUs/IO/Drives/SoE/Ax5000ParamSTRUCTs/P/AX5000_P_0020.TcDUT
TYPE AX5000_P_0020 :
STRUCT
	EhterCAT_device_identification:UINT:=1;
END_STRUCT
END_TYPE

// ---- POUs/IO/Drives/SoE/Ax5000ParamSTRUCTs/P/AX5000_P_0050.TcDUT
TYPE AX5000_P_0050 :
STRUCT
	Funktional_principle:INT;
	Construktion:INT;
	revd:ARRAY[0..14] OF UINT;

END_STRUCT
END_TYPE

// ---- POUs/IO/Drives/SoE/Ax5000ParamSTRUCTs/P/AX5000_P_0051.TcDUT
TYPE AX5000_P_0051 :
STRUCT
	Number_of_pole_pairs:UINT;
END_STRUCT
END_TYPE

// ---- POUs/IO/Drives/SoE/Ax5000ParamSTRUCTs/P/AX5000_P_0053.TcDUT
TYPE AX5000_P_0053 :
STRUCT
	Actual_lenght:UINT;
	Max_lenght:UINT;
	Configures_motor_type:STRING(29);

END_STRUCT
END_TYPE

// ---- POUs/IO/Drives/SoE/Ax5000ParamSTRUCTs/P/AX5000_P_0056.TcDUT
TYPE AX5000_P_0056 :
STRUCT
	Max_motor_speed_with_max_torque:UDINT;
END_STRUCT
END_TYPE

// ---- POUs/IO/Drives/SoE/Ax5000ParamSTRUCTs/P/AX5000_P_0057.TcDUT
TYPE AX5000_P_0057 :
STRUCT
	Electrical_commutation_offset:UINT;
END_STRUCT
END_TYPE

// ---- POUs/IO/Drives/SoE/Ax5000ParamSTRUCTs/P/AX5000_P_0059.TcDUT
TYPE AX5000_P_0059 :
STRUCT
	Motor_brake_current_monitoring_level:UINT;
END_STRUCT
END_TYPE

// ---- POUs/IO/Drives/SoE/Ax5000ParamSTRUCTs/P/AX5000_P_0061.TcDUT
TYPE AX5000_P_0061 :
STRUCT
	Motor_temperature_sensor_type:UINT;
END_STRUCT
END_TYPE

// ---- POUs/IO/Drives/SoE/Ax5000ParamSTRUCTs/P/AX5000_P_0065.TcDUT
TYPE AX5000_P_0065 :
STRUCT
	Actual_temperature_sensor_resistance:UINT;
END_STRUCT
END_TYPE

// ---- POUs/IO/Drives/SoE/Ax5000ParamSTRUCTs/P/AX5000_P_0067.TcDUT
TYPE AX5000_P_0067 :
STRUCT
	Motor_winding_dielektric_strength:UINT;
END_STRUCT
END_TYPE

// ---- POUs/IO/Drives/SoE/Ax5000ParamSTRUCTs/P/AX5000_P_0070.TcDUT
TYPE AX5000_P_0070 :
STRUCT
	Motor_contunuouse_stall_torque:UINT;
END_STRUCT
END_TYPE

// ---- POUs/IO/Drives/SoE/Ax5000ParamSTRUCTs/P/AX5000_P_0078.TcDUT
TYPE AX5000_P_0078 :
STRUCT
	Max_motor_dc_link_voltage:UINT;
END_STRUCT
END_TYPE

// ---- POUs/IO/Drives/SoE/Ax5000ParamSTRUCTs/P/AX5000_P_0088.TcDUT
TYPE AX5000_P_0088 :
STRUCT
	Velocity_limit_value:UDINT;
	Corresponding_current_value:UINT;
END_STRUCT
END_TYPE

// ---- POUs/IO/Drives/SoE/Ax5000ParamSTRUCTs/P/AX5000_P_0093.TcDUT
TYPE AX5000_P_0093 :
STRUCT
	Configures_channel_current:UDINT;
END_STRUCT
END_TYPE

// ---- POUs/IO/Drives/SoE/Ax5000ParamSTRUCTs/P/AX5000_P_0097.TcDUT
TYPE AX5000_P_0097 :
STRUCT
	Motor_brake_unlocked:BOOL;
	Rsvd:ARRAY[0..14] OF BOOL;
END_STRUCT
END_TYPE

// ---- POUs/IO/Drives/SoE/Ax5000ParamSTRUCTs/P/AX5000_P_0110.TcDUT
TYPE AX5000_P_0110 :
STRUCT
	ASM_motor_magnetzing_inductance:UDINT;
END_STRUCT
END_TYPE

// ---- POUs/IO/Drives/SoE/Ax5000ParamSTRUCTs/P/AX5000_P_0114.TcDUT
TYPE AX5000_P_0114 :
STRUCT
	ASM_acceleration_control_integral_action_time:UINT;
END_STRUCT
END_TYPE

// ---- POUs/IO/Drives/SoE/Ax5000ParamSTRUCTs/P/AX5000_P_0119.TcDUT
TYPE AX5000_P_0119 :
STRUCT
	ASM_boost_voltage_slope:UDINT;
END_STRUCT
END_TYPE

// ---- POUs/IO/Drives/SoE/Ax5000ParamSTRUCTs/P/AX5000_P_0152.TcDUT
TYPE AX5000_P_0152 :
STRUCT
	Feedback_1_geat_numerator:UDINT;
END_STRUCT
END_TYPE

// ---- POUs/IO/Drives/SoE/Ax5000ParamSTRUCTs/P/AX5000_P_0154.TcDUT
TYPE AX5000_P_0154 :
STRUCT
	Actual_lenght:UINT;
	Max_lenght:UINT;
	Reference_source:UINT;
	Reference_index:UINT;
	Threshold_voltage:UINT;
//{attribute 'hide'}
	rsvd:UINT;
END_STRUCT
END_TYPE

// ---- POUs/IO/Drives/SoE/Ax5000ParamSTRUCTs/P/AX5000_P_0158.TcDUT
TYPE AX5000_P_0158 :
STRUCT
	Save_feedback_identication:UINT;
END_STRUCT
END_TYPE

// ---- POUs/IO/Drives/SoE/Ax5000ParamSTRUCTs/P/AX5000_P_0159.TcDUT
TYPE AX5000_P_0159 :
STRUCT
	Raw_position_feedback_value:UDINT;
END_STRUCT
END_TYPE

// ---- POUs/IO/Drives/SoE/Ax5000ParamSTRUCTs/P/AX5000_P_0162.TcDUT
TYPE AX5000_P_0162 :
STRUCT
	Feedback1_save_digital_nameplate:UINT;
END_STRUCT
END_TYPE

// ---- POUs/IO/Drives/SoE/Ax5000ParamSTRUCTs/P/AX5000_P_0166.TcDUT
TYPE AX5000_P_0166 :
STRUCT
	Motor_and_feedback_connection_ceck:UINT;
END_STRUCT
END_TYPE

// ---- POUs/IO/Drives/SoE/Ax5000ParamSTRUCTs/P/AX5000_P_0169.TcDUT
{attribute 'pack_mode' := '1'}//Ensures 1-byte-alignmend
TYPE AX5000_P_0169 :
STRUCT
	Actual_lenght:UINT;
	Max_lenght:UINT;
(*Onboard*)
	DelayRegister:UINT;
	QualityMonitorValue:UINT;
	SlaveRSSI:UINT;
	EdgeRegister:UINT;
	SummaryRegister:UINT;
	EncoderTemperature:INT;
	LEDCurrent:UINT;
	SupplyVoltage:UINT;
	EncoderStatus0:USINT;
	EncoderStatus1:USINT;
	EncoderStatus2:USINT;
	EncoderStatus3:USINT;
	EncoderStatus4:USINT;
	EncoderStatus5:USINT;
	EncoderStatus6:USINT;
	EncoderStatus7:USINT;
	EncoderStatus0_detailed:USINT;
	EncoderStatus1_detailed:USINT;
	EncoderStatus2_detailed:USINT;
	EncoderStatus3_detailed:USINT;
	EncoderStatus4_detailed:USINT;
	EncoderStatus5_detailed:USINT;
	EncoderStatus6_detailed:USINT;
	EncoderStatus7_detailed:USINT;
	OperatingTime:UDINT;
	TotalShaftTurns:UDINT;
//{attribute 'hide'}
	Rsvd:ARRAY[0..2] OF UINT;
	MaxOccuredPositionDelivation:UINT;
	TotalVPOSErrors:UINT;
	TotalACCErrors:UINT;
	TotalPOSErrors:UINT;
	TotalLINKErrors:UINT;
	TotalEncodingErrors:UINT;
//{attribute 'hide'}
	Rsvd2:UINT;
//{attribute 'hide'}
	Rsvd3:UINT;
	CyclicReadCounter:UINT;
	CyclicReadErrorCounter:UINT;


(*AX57xx*)			(*Die beiden NICHT verwendeten Feedbacksystemeauf der AX57xx müssen ausgeklammert werden*)

		(*HiperfaceDSL
			DelayRegister:UINT;
			QualityMonitorValue:UINT;
			SlaveRSSI:UINT;
			EdgeRegister:UINT;
			SummaryRegister:UINT;
			EncoderTemperature:INT;
			LEDCurrent:UINT;
			SupplyVoltage:UINT;
			EncoderStatus0:USINT;
			EncoderStatus1:USINT;
			EncoderStatus2:USINT;
			EncoderStatus3:USINT;
			EncoderStatus4:USINT;
			EncoderStatus5:USINT;
			EncoderStatus6:USINT;
			EncoderStatus7:USINT;
			EncoderStatus0_detailed:USINT;
			EncoderStatus1_detailed:USINT;
			EncoderStatus2_detailed:USINT;
			EncoderStatus3_detailed:USINT;
			EncoderStatus4_detailed:USINT;
			EncoderStatus5_detailed:USINT;
			EncoderStatus6_detailed:USINT;
			EncoderStatus7_detailed:USINT;
			OperatingTime:UDINT;
			TotalShaftTurns:UDINT;
	//	{attribute 'hide'}
			rsvd:ARRAY[0..2] OF UINT;
			MaxOccuredPositionDelivation:UINT;
			TotalVPOSErrors:UINT;
			TotalACCErrors:UINT;
			TotalPOSErrors:UINT;
			TotalLINKErrors:UINT;
			TotalEncodingErrors:UINT;
		//	{attribute 'hide'}
			rsvd2:UINT;
		//	{attribute 'hide'}
			rsvd3:UINT;
			CyclicReadCounter:UINT;
			CyclicReadErrorCounter:UINT;
*)
(*

		(*AX572xEnDat2.2*)

			AX572xEnDat2.2:UINT;

*)

(*
		(*AX572xBiSS*)

			AX572xBiSS:UINT;
*)

END_STRUCT
END_TYPE

// ---- POUs/IO/Drives/SoE/Ax5000ParamSTRUCTs/P/AX5000_P_0188.TcDUT
TYPE AX5000_P_0188 :
STRUCT
	Save_feedback_identication:UINT;
END_STRUCT
END_TYPE

// ---- POUs/IO/Drives/SoE/Ax5000ParamSTRUCTs/P/AX5000_P_0196.TcDUT
TYPE AX5000_P_0196 :
STRUCT
	Actual_lenght:UINT;
	Max_lenght:UINT;
	Numeration:UDINT;
	Denominator:UDINT;
	Mask:UDINT;
	Position_offset:UDINT;
	Data_valid:UINT;
//	{attribute 'hide'}
	rsvd:UINT;
END_STRUCT
END_TYPE

// ---- POUs/IO/Drives/SoE/Ax5000ParamSTRUCTs/P/AX5000_P_0205.TcDUT
TYPE AX5000_P_0205 :
STRUCT
	Power_management_status_word:UINT;
END_STRUCT
END_TYPE

// ---- POUs/IO/Drives/SoE/Ax5000ParamSTRUCTs/P/AX5000_P_0207.TcDUT
{attribute 'pack_mode' := '1'}//Ensures 1-byte-alignmend
TYPE AX5000_P_0207 :
STRUCT
	Actual_lenght:UINT;
	Max_lenght:UINT;
	Resistance:UINT;
	Continuous_Power:UINT;
	Period_time_for_duty_cycle:UINT;
	Brake_resistor_protection:UINT;
	Maximum_peak_energy_by_40Percent_duty_cycle:UDINT;
	Maximum_peak_energy_by_20Percent_duty_cycle:UDINT;
	Maximum_peak_energy_by_10Percent_duty_cycle:UDINT;
	Maximum_peak_energy_by_1Percent_duty_cycle:UDINT;
	Maximum_peak_energy_by_01Percent_duty_cycle:UDINT;
	Rsvd:ARRAY[0..3] OF UDINT;

END_STRUCT
END_TYPE

// ---- POUs/IO/Drives/SoE/Ax5000ParamSTRUCTs/P/AX5000_P_0208.TcDUT
{attribute 'pack_mode' := '1'}//Ensures 1-byte-alignmend
TYPE AX5000_P_0208 :
STRUCT
	Actual_lenght:UINT;
	Max_lenght:UINT;
	Resistance:UINT;
	Continuous_Power:UINT;
	Period_time_for_duty_cycle:UINT;
	Brake_resistor_protection:UINT;
	Maximum_peak_energy_by_40Percent_duty_cycle:UDINT;
	Maximum_peak_energy_by_20Percent_duty_cycle:UDINT;
	Maximum_peak_energy_by_10Percent_duty_cycle:UDINT;
	Maximum_peak_energy_by_1Percent_duty_cycle:UDINT;
	Maximum_peak_energy_by_01Percent_duty_cycle:UDINT;
	Rsvd:ARRAY[0..3] OF UDINT;

END_STRUCT
END_TYPE

// ---- POUs/IO/Drives/SoE/Ax5000ParamSTRUCTs/P/AX5000_P_0212.TcDUT
TYPE AX5000_P_0212 :
STRUCT
	Warning_level_Actual_cont_power_external_brake_resistor:UINT;
END_STRUCT
END_TYPE

// ---- POUs/IO/Drives/SoE/Ax5000ParamSTRUCTs/P/AX5000_P_0213.TcDUT
TYPE AX5000_P_0213 :
STRUCT
	External_DC_Link_current:DINT;
END_STRUCT
END_TYPE

// ---- POUs/IO/Drives/SoE/Ax5000ParamSTRUCTs/P/AX5000_P_0215.TcDUT
TYPE AX5000_P_0215 :
STRUCT
	Actual_Periphery_Voltage:UINT;
END_STRUCT
END_TYPE

// ---- POUs/IO/Drives/SoE/Ax5000ParamSTRUCTs/P/AX5000_P_0219.TcDUT
TYPE AX5000_P_0219 :
STRUCT
	External_brake_resistor_actual_peak_energy:UINT;
END_STRUCT
END_TYPE

// ---- POUs/IO/Drives/SoE/Ax5000ParamSTRUCTs/P/AX5000_P_0251.TcDUT
TYPE AX5000_P_0251 EXTENDS ST_AX5000_P_0251:
STRUCT
(*	Actual_lenght:UINT;
	Max_lenght:UINT;
	Mux1:UINT;
	Mux2:UINT;
	Logic:UINT;
	Latch_ctrl:UINT;
*)
END_STRUCT
END_TYPE

// ---- POUs/IO/Drives/SoE/Ax5000ParamSTRUCTs/P/AX5000_P_0252.TcDUT
TYPE AX5000_P_0252 :
STRUCT
	Probe_1_logic_state:UINT;
END_STRUCT
END_TYPE

// ---- POUs/IO/Drives/SoE/Ax5000ParamSTRUCTs/P/AX5000_P_0253.TcDUT
TYPE AX5000_P_0253 :
STRUCT
	Probe_1_time_positive_edge:UDINT;
END_STRUCT
END_TYPE

// ---- POUs/IO/Drives/SoE/Ax5000ParamSTRUCTs/P/AX5000_P_0255.TcDUT
TYPE AX5000_P_0255 :
STRUCT
	Probe_1_timer_difference_reference_switch_to_index:UDINT;
END_STRUCT
END_TYPE

// ---- POUs/IO/Drives/SoE/Ax5000ParamSTRUCTs/P/AX5000_P_0256.TcDUT
{attribute 'pack_mode' := '1'}//Ensures 1-byte-alignmend
TYPE AX5000_P_0256 :
STRUCT
	Actual_lenght:UINT;
	Max_lenght:UINT;
(*Positive Edge*)
	Times:ARRAY[0..1] OF UDINT;
	Values:ARRAY[0..1] OF UDINT;
	Rsvd1:ARRAY[0..1] OF UDINT;
	Last_time_index:UINT;
	Last_value_index:UINT;
	Latched_time:UDINT;
	Latched_value:UDINT;
(*Negative Edge*)
	Times2:ARRAY[0..1] OF UDINT;
	Values2:ARRAY[0..1] OF UDINT;
	Rsvd2:ARRAY[0..1] OF UDINT;
	Last_time_index2:UINT;
	Last_value_index2:UINT;
	Latched_time2:UDINT;
	Latched_value2:UDINT;
END_STRUCT
END_TYPE

// ---- POUs/IO/Drives/SoE/Ax5000ParamSTRUCTs/P/AX5000_P_0273.TcDUT
TYPE AX5000_P_0273 EXTENDS ST_AX5000_P_0273:
STRUCT
(*
	Actual_lenght:UINT:= 112;
	Max_lenght:UINT := 112;
(*feedback 1*)
 {attribute 'GUID' := 'D1EB669D-3061-44CC-A2EE-FBF75E3AC2F6'}
 {attribute 'Namespace' := 'AX5000'}
Feedback1 : ST_AX5000_P_0273_Feedback;
(*
(*Encoder Memory*)
	Data_valid1:UINT;
//	{attribute 'hide'}
	rsvd1:UINT;
	Position_offset1:UDINT;
(*Drive Memory*)
	Data_valid2:UINT;
//	{attribute 'hide'}
	rsvd2:UINT;
	Feedback_type1:STRING(29);
//	{attribute 'hide'}
	rsvd3:UINT;
	Feedback_serial_number:ARRAY[0..1]OF UDINT;
	Position_offset2:UDINT;
*)
(*feedback 2*)
{attribute 'GUID' := 'D1EB669D-3061-44CC-A2EE-FBF75E3AC2F6'}
 {attribute 'Namespace' := 'AX5000'}
Feedback2 : ST_AX5000_P_0273_Feedback;
(*
(*Encoder Memory*)
	Data_valid3:UINT;
//	{attribute 'hide'}
	rsvd4:UINT;
	Position_offset3:UDINT;
(*Drive Memory*)
	Data_valid4:UINT;
//	{attribute 'hide'}
	rsvd5:UINT;
	Feedback_type2:STRING(29);
//	{attribute 'hide'}
	rsvd6:UINT;
	Feedback_serial_number2:ARRAY[0..1]OF UDINT;
	Position_offset4:UDINT;
*)	

//	{attribute 'hide'}
	Rsvd1 : UDINT;
*)
END_STRUCT
END_TYPE

// ---- POUs/IO/Drives/SoE/Ax5000ParamSTRUCTs/P/AX5000_P_0275.TcDUT
TYPE AX5000_P_0275 EXTENDS ST_AX5000_P_0275: 
	STRUCT
(*		 {attribute 'GUID' := 'A39361D3-D4AC-4F67-8FEE-F366F3137B89'}
		 {attribute 'Namespace' := 'AX5000'}
		ActiveFeedbackAndMemory : E_AX5000_P_0275_ActiveFeedbackAndMemory;
		InitializationErrorBehavior : BIT;
		 {attribute 'hide'}
		_reserved1 : BIT;
		 {attribute 'hide'}
		_reserved2 : BIT;
		 {attribute 'hide'}
		_reserved3 : BIT;
		 {attribute 'hide'}
		_reserved4 : BIT;
		 {attribute 'hide'}
		_reserved5 : BIT;
		 {attribute 'hide'}
		_reserved6 : BIT;
		 {attribute 'hide'}
		_reserved7 : BIT;
*)
	END_STRUCT
END_TYPE

// ---- POUs/IO/Drives/SoE/Ax5000ParamSTRUCTs/P/AX5000_P_0301.TcDUT
TYPE AX5000_P_0301 :
STRUCT
	Actual_lenght:UINT;
	Max_lenght:UINT;
	Error_times_history:ARRAY[0..99] OF UDINT;
END_STRUCT
END_TYPE

// ---- POUs/IO/Drives/SoE/Ax5000ParamSTRUCTs/P/AX5000_P_0304.TcDUT
TYPE AX5000_P_0304 :
STRUCT
	Log_errors_Log_warnings_Log_information_rsvd:UINT;	(*Log_errors 1; BitLog_warnings 1; BitLog_information 1 Bit*)
END_STRUCT
END_TYPE

// ---- POUs/IO/Drives/SoE/Ax5000ParamSTRUCTs/P/AX5000_P_0308.TcDUT
TYPE AX5000_P_0308 :
STRUCT
	Actual_ctrl_loop_time:UINT;
END_STRUCT
END_TYPE

// ---- POUs/IO/Drives/SoE/Ax5000ParamSTRUCTs/P/AX5000_P_0310.TcDUT
TYPE AX5000_P_0310 :
STRUCT
	Torque_off_Slow_down_according_Open_loop_ramp_Closed_loop_ramp_NC_handling_rsvd:UINT;
	(*Torque_off 1 Bit; Slow_down_according 1 Bit; Open_loop_ramp 1 Bit; Closed_loop_ramp 1 Bit; NC_handling  1 Bit;  rsvd  11 Bit; *)
END_STRUCT
END_TYPE

// ---- POUs/IO/Drives/SoE/Ax5000ParamSTRUCTs/P/AX5000_P_0312.TcDUT
TYPE AX5000_P_0312 :
STRUCT
	PCB_temperature:UINT;
END_STRUCT
END_TYPE

// ---- POUs/IO/Drives/SoE/Ax5000ParamSTRUCTs/P/AX5000_P_0314.TcDUT
TYPE AX5000_P_0314 :
STRUCT
	Actual_lenght:UINT;
	Max_lenght:UINT;
	String_output_mode:UINT;
	Backlight_mode:UINT;
	Keypad_mode:UINT;
//	{attribute 'hide'}
	Rsvd:UINT;
	Output_string:STRING(39);
END_STRUCT
END_TYPE

// ---- POUs/IO/Drives/SoE/Ax5000ParamSTRUCTs/P/AX5000_P_0315.TcDUT
TYPE AX5000_P_0315 :
STRUCT
	Configuration_Output_number_Set_output_error_Set_output_warning_rsvd:UINT;
	(*Configuration 3 Bit; Output_number 5 Bit; Set_output_error 1 Bit; Set_output_warning 1 Bit; rsvd 6 Bit; *)
END_STRUCT
END_TYPE

// ---- POUs/IO/Drives/SoE/Ax5000ParamSTRUCTs/P/AX5000_P_0316.TcDUT
TYPE AX5000_P_0316 :
STRUCT
	Actual_lenght:UINT;
	Max_lenght:UINT;
	Mode:UINT;
	Level:UINT;		(*Decimal Point 1*)
END_STRUCT
END_TYPE

// ---- POUs/IO/Drives/SoE/Ax5000ParamSTRUCTs/P/AX5000_P_0323.TcDUT
TYPE AX5000_P_0323 :
STRUCT
	Actual_lenght:UINT;
	Max_lenght:UINT;

(*control*)
	Total:UDINT;
	Available:UDINT;
	Total1:UDINT;
	Available1:UDINT;
	Total2:UDINT;
	Available2:UDINT;
	Total3:UDINT;
	Available3:UDINT;

(*front*)
	Total4:UDINT;
	Available4:UDINT;
	Total5:UDINT;
	Available5:UDINT;
	Total6:UDINT;
	Available6:UDINT;
	Total7:UDINT;
	Available7:UDINT;


(*option*)
	Toal8:UDINT;
	Available8:UDINT;
	Total9:UDINT;
	Available9:UDINT;
	Total10:UDINT;
	Available10:UDINT;
	Total11:UDINT;
	Available11:UDINT;
END_STRUCT
END_TYPE

// ---- POUs/IO/Drives/SoE/Ax5000ParamSTRUCTs/P/AX5000_P_0350.TcDUT
TYPE AX5000_P_0350 EXTENDS ST_AX5000_P_0350: 
STRUCT
//	Error_reaction_Controlword:UINT;
END_STRUCT
END_TYPE

// ---- POUs/IO/Drives/SoE/Ax5000ParamSTRUCTs/P/AX5000_P_0356.TcDUT
//	{attribute 'hide'}
TYPE AX5000_P_0356 :
STRUCT
	Actual_lenght:UINT;
	Max_lenght:UINT;
//	{attribute 'hide'}
	Rsvd:UDINT;
	Available_for:UINT;
	Command_mode:UINT;
	Current_level:UINT;
	Current_slope:UINT;
	Wait_time_before_braking:UINT;
	First_phase_activation_time_with_f_f1:UINT;
	Rotary_field_frequency_f1:UINT;
	Rotor_slowdown_mode:UINT;
	Second_phase_activation_time_with_f_0Hz:UINT;
	Wait_ime_after_braking:UINT;
//	{attribute 'hide'}
	Rsvd1:UINT;
//	{attribute 'hide'}
	Rsvd2:UINT;
	Synchronus_motor:ARRAY[0..11] OF UINT;
END_STRUCT
END_TYPE

// ---- POUs/IO/Drives/SoE/Ax5000ParamSTRUCTs/P/AX5000_P_0360.TcDUT
TYPE AX5000_P_0360 :
STRUCT
	Parameter_set_prearrangement:UINT;
END_STRUCT
END_TYPE

// ---- POUs/IO/Drives/SoE/Ax5000ParamSTRUCTs/P/AX5000_P_0402.TcDUT
TYPE AX5000_P_0402 :
STRUCT
	Redy_to_operate_configuration:UINT;
END_STRUCT
END_TYPE

// ---- POUs/IO/Drives/SoE/Ax5000ParamSTRUCTs/P/AX5000_P_0451.TcDUT
TYPE AX5000_P_0451 :
STRUCT
	Current_controller_settings:UINT;
END_STRUCT
END_TYPE

// ---- POUs/IO/Drives/SoE/Ax5000ParamSTRUCTs/P/AX5000_P_0457.TcDUT
TYPE AX5000_P_0457 :
STRUCT
	Actual_motor_voltage_phase_V:UINT;
END_STRUCT
END_TYPE

// ---- POUs/IO/Drives/SoE/Ax5000ParamSTRUCTs/P/AX5000_P_0459.TcDUT
TYPE AX5000_P_0459 :
STRUCT
	Actual_torquw_generating_current:UINT;
END_STRUCT
END_TYPE

// ---- POUs/IO/Drives/SoE/Ax5000ParamSTRUCTs/P/AX5000_P_0461.TcDUT
TYPE AX5000_P_0461 :
STRUCT
	Actual_absolute_current:UINT;
END_STRUCT
END_TYPE

// ---- POUs/IO/Drives/SoE/Ax5000ParamSTRUCTs/P/AX5000_P_0504.TcDUT
TYPE AX5000_P_0504 :
STRUCT
	Effective_velocity_command_value:UDINT;
END_STRUCT
END_TYPE

// ---- POUs/IO/Drives/SoE/Ax5000ParamSTRUCTs/P/AX5000_P_0511.TcDUT
TYPE AX5000_P_0511 :
STRUCT
	Celocity_filter_low_pass_time_constant:UINT;
END_STRUCT
END_TYPE

// ---- POUs/IO/Drives/SoE/Ax5000ParamSTRUCTs/P/AX5000_P_0515.TcDUT
{attribute 'pack_mode' := '1'}
TYPE AX5000_P_0515 :
STRUCT
	Actual_lenght:UINT;
	Max_lenght:UINT;
	ST_CONV_Version:UINT;
//	{attribute 'hide'}
	Rsvd1:UINT;
	Filter_type:UINT;
//	{attribute 'hide'}
	Rsvd2:UINT;
	Low_pass_frequency:UDINT;
	Low_pass_damping:UDINT;
	High_pass_frequency:UDINT;
	High_pass_damping:UDINT;
//	{attribute 'hide'}
	Rsvd3:UDINT;
//	{attribute 'hide'}
	Rsvd4:UDINT;
	QMath_factor:UINT;
//	{attribute 'hide'}
	Rsvd5:UINT;
	b0:UDINT;
	b1:UDINT;
	b2:UDINT;
	a1:UDINT;
	a2:UDINT;
//	{attribute 'hide'}
	Rsvd6:UDINT;
//	{attribute 'hide'}
	Rsvd7:UDINT;
END_STRUCT
END_TYPE

// ---- POUs/IO/Drives/SoE/Ax5000ParamSTRUCTs/P/AX5000_P_0517.TcDUT
{attribute 'pack_mode' := '1'}
TYPE AX5000_P_0517 :
STRUCT
	Actual_lenght:UINT;
	Max_lenght:UINT;
	ST_CONV_Version:UINT;
//	{attribute 'hide'}
	Rsvd1:UINT;
	Filter_type:UINT;
//	{attribute 'hide'}
	Rsvd2:UINT;
	Low_pass_frequency:UDINT;
	Low_pass_damping:UDINT;
	High_pass_frequency:UDINT;
	High_pass_damping:UDINT;
//	{attribute 'hide'}
	Rsvd3:UDINT;
//	{attribute 'hide'}
	nRsvd4:UDINT;
	QMath_factor:UINT;
	Rsvd5:UINT;
	b0:UDINT;
	b1:UDINT;
	b2:UDINT;
	a1:UDINT;
	a2:UDINT;
//	{attribute 'hide'}
	Rsvd6:UDINT;
//	{attribute 'hide'}
	Rsvd7:UDINT;
END_STRUCT
END_TYPE

// ---- POUs/IO/Drives/SoE/Ax5000ParamSTRUCTs/P/AX5000_P_0518.TcDUT
{attribute 'pack_mode' := '1'}
TYPE AX5000_P_0518 :
STRUCT
	Actual_lenght:UINT;
	Max_lenght:UINT;
	Mode:UINT;
//	{attribute 'hide'}
	Rsvd:UINT;
	Velocity_window:UDINT;
	TIME_:UINT;
//	{attribute 'hide'}
	Rsvd1:UINT;
//	{attribute 'hide'}
	Rsvd2:UINT;
//	{attribute 'hide'}
	Rsvd3:UINT;
END_STRUCT
END_TYPE

// ---- POUs/IO/Drives/SoE/Ax5000ParamSTRUCTs/P/AX5000_P_0553.TcDUT
TYPE AX5000_P_0553 :
STRUCT
	Position_controller_status_word:UINT;
END_STRUCT
END_TYPE

// ---- POUs/IO/Drives/SoE/Ax5000ParamSTRUCTs/P/AX5000_P_0554.TcDUT
TYPE AX5000_P_0554 :
STRUCT
	Effective_position_command_value:DINT;
END_STRUCT
END_TYPE

// ---- POUs/IO/Drives/SoE/Ax5000ParamSTRUCTs/P/AX5000_P_0601.TcDUT
TYPE AX5000_P_0601 :
STRUCT
	Predictive_velocity_command_value:DINT;
END_STRUCT
END_TYPE

// ---- POUs/IO/Drives/SoE/Ax5000ParamSTRUCTs/P/AX5000_P_0801.TcDUT
TYPE AX5000_P_0801 :
STRUCT
	Digital_inputs_state:UINT;
END_STRUCT
END_TYPE

// ---- POUs/IO/Drives/SoE/Ax5000ParamSTRUCTs/P/AX5000_P_0806.TcDUT
TYPE AX5000_P_0806 :
STRUCT
	Amplifier_output_voltage_slope:INT;
END_STRUCT
END_TYPE

// ---- POUs/IO/Drives/SoE/Ax5000ParamSTRUCTs/P/AX5000_P_0850.TcDUT
TYPE AX5000_P_0850 :
STRUCT
	Actual_lenght:UINT;
	Max_lenght:UINT;
	Amplifier_identification:STRING(63);
END_STRUCT
END_TYPE

// ---- POUs/IO/Drives/SoE/Ax5000ParamSTRUCTs/P/AX5000_P_0851.TcDUT
TYPE AX5000_P_0851 :
STRUCT
	Save_amplifier_identification:UINT;
END_STRUCT
END_TYPE

// ---- POUs/IO/Drives/SoE/Ax5000ParamSTRUCTs/P/AX5000_P_0902.TcDUT
TYPE AX5000_P_0902 :
STRUCT
	Current_calibration:UINT;
END_STRUCT
END_TYPE

// ---- POUs/IO/Drives/SoE/Ax5000ParamSTRUCTs/P/AX5000_P_0912.TcDUT
TYPE AX5000_P_0912 :
STRUCT
	Actual_lenght:UINT;
	Max_lenght:UINT;
	Calibration:UINT;
	Calibration_type:UINT;
	Calibration_point:UINT;
	Calibration_current:UINT;
	Calibration_phase:UINT;
	Calibration_tolerance:UINT;
END_STRUCT
END_TYPE

// ---- POUs/IO/Drives/SoE/Ax5000ParamSTRUCTs/P/AX5000_P_1001.TcDUT
TYPE AX5000_P_1001 :
STRUCT
	Debug_pointer_1_typ:UINT;
END_STRUCT
END_TYPE

// ---- POUs/IO/Drives/SoE/Ax5000ParamSTRUCTs/P/AX5000_P_1007.TcDUT
TYPE AX5000_P_1007 :
STRUCT
	Feedback_debug_pointer_1_typ:UINT;
END_STRUCT
END_TYPE

// ---- POUs/IO/Drives/SoE/Ax5000ParamSTRUCTs/P/AX5000_P_1008.TcDUT
TYPE AX5000_P_1008 :
STRUCT
	Feedback_debug_pointer_1_value:UINT;
END_STRUCT
END_TYPE

// ---- POUs/IO/Drives/SoE/Ax5000ParamSTRUCTs/P/AX5000_P_1022.TcDUT
TYPE AX5000_P_1022 :
STRUCT
	Deburg_command:UINT;
END_STRUCT
END_TYPE

// ---- POUs/IO/Drives/SoE/Ax5000ParamSTRUCTs/P/AX5000_P_2000.TcDUT
TYPE AX5000_P_2000 :
STRUCT
	Configured_safety_option: E_AX5000_P_2000_SafetyOption;
END_STRUCT
END_TYPE

// ---- POUs/IO/Drives/SoE/Ax5000ParamSTRUCTs/P/AX5000_P_2001.TcDUT
TYPE AX5000_P_2001 :
STRUCT
	Safety_option_diagnostics:UINT;
END_STRUCT
END_TYPE

// ---- POUs/IO/Drives/SoE/Ax5000ParamSTRUCTs/P/AX5000_P_2002.TcDUT
TYPE AX5000_P_2002 :
STRUCT
	Safety_option_state:UINT;
END_STRUCT
END_TYPE

// ---- POUs/IO/Drives/SoE/Ax5000ParamSTRUCTs/S/AX5000_S_0001.TcDUT
TYPE AX5000_S_0001 :
STRUCT
	Switching_frequency_of_the_IGBT_module:UINT;
END_STRUCT
END_TYPE

// ---- POUs/IO/Drives/SoE/Ax5000ParamSTRUCTs/S/AX5000_S_0011.TcDUT
TYPE AX5000_S_0011 :
STRUCT
	Class_1_diagnostic:UINT;
END_STRUCT
END_TYPE

// ---- POUs/IO/Drives/SoE/Ax5000ParamSTRUCTs/S/AX5000_S_0013.TcDUT
TYPE AX5000_S_0013 :
STRUCT
	Class_3_diagnostic:UINT;
END_STRUCT
END_TYPE

// ---- POUs/IO/Drives/SoE/Ax5000ParamSTRUCTs/S/AX5000_S_0015.TcDUT
TYPE AX5000_S_0015 :
STRUCT
	Telefram_type:UINT;
END_STRUCT
END_TYPE

// ---- POUs/IO/Drives/SoE/Ax5000ParamSTRUCTs/S/AX5000_S_0018.TcDUT
TYPE AX5000_S_0018 :
STRUCT
	Actual_lenght:UINT;
	Max_lenght:UINT;
	IDN_list_of_all_operation_data_for_CP2: ARRAY[0..346] OF UINT;
END_STRUCT
END_TYPE

// ---- POUs/IO/Drives/SoE/Ax5000ParamSTRUCTs/S/AX5000_S_0030.TcDUT
TYPE AX5000_S_0030 :
STRUCT
	Actual_lenght:UINT;
	Max_lenght:UINT;
	Manufacturer_version:STRING(61);
END_STRUCT
END_TYPE

// ---- POUs/IO/Drives/SoE/Ax5000ParamSTRUCTs/S/AX5000_S_0031.TcDUT
TYPE AX5000_S_0031 :
STRUCT
	Actual_lenght:UINT;
	Max_lenght:UINT;
	Hardware_version:STRING(45)
;END_STRUCT
END_TYPE

// ---- POUs/IO/Drives/SoE/Ax5000ParamSTRUCTs/S/AX5000_S_0037.TcDUT
TYPE AX5000_S_0037 :
STRUCT
	Additive_Velocity_command_value:DINT;
END_STRUCT
END_TYPE

// ---- POUs/IO/Drives/SoE/Ax5000ParamSTRUCTs/S/AX5000_S_0048.TcDUT
TYPE AX5000_S_0048 :
STRUCT
	Additive_position_command_value:DINT;
END_STRUCT
END_TYPE

// ---- POUs/IO/Drives/SoE/Ax5000ParamSTRUCTs/S/AX5000_S_0053.TcDUT
TYPE AX5000_S_0053 :
STRUCT
	Position_feedback_value_2:DINT;
END_STRUCT
END_TYPE

// ---- POUs/IO/Drives/SoE/Ax5000ParamSTRUCTs/S/AX5000_S_0080.TcDUT
TYPE AX5000_S_0080 :
STRUCT
	Torque_command_value:INT;
END_STRUCT
END_TYPE

// ---- POUs/IO/Drives/SoE/Ax5000ParamSTRUCTs/S/AX5000_S_0081.TcDUT
TYPE AX5000_S_0081 :
STRUCT
	Additive_Torque_command_value:INT;
END_STRUCT
END_TYPE

// ---- POUs/IO/Drives/SoE/Ax5000ParamSTRUCTs/S/AX5000_S_0086.TcDUT
TYPE AX5000_S_0086 :
STRUCT
	Torque_force_data_scaling_type:UINT;
END_STRUCT
END_TYPE

// ---- POUs/IO/Drives/SoE/Ax5000ParamSTRUCTs/S/AX5000_S_0091.TcDUT
TYPE AX5000_S_0091 :
STRUCT
	Bipolar_velocity_limit_value:UDINT;
END_STRUCT
END_TYPE

// ---- POUs/IO/Drives/SoE/Ax5000ParamSTRUCTs/S/AX5000_S_0095.TcDUT
TYPE AX5000_S_0095 :
STRUCT
	Actual_lenght:UINT;
	Max_lenght:UINT;
	Diagnistic_message:STRING(99);
END_STRUCT
END_TYPE

// ---- POUs/IO/Drives/SoE/Ax5000ParamSTRUCTs/S/AX5000_S_0099.TcDUT
TYPE AX5000_S_0099 :
STRUCT
	Reset_class_1_diagnistic:UINT;
END_STRUCT
END_TYPE

// ---- POUs/IO/Drives/SoE/Ax5000ParamSTRUCTs/S/AX5000_S_0100.TcDUT
TYPE AX5000_S_0100 :
STRUCT
	Velocity_loop_proportional_gain:UDINT;
END_STRUCT
END_TYPE

// ---- POUs/IO/Drives/SoE/Ax5000ParamSTRUCTs/S/AX5000_S_0104.TcDUT
TYPE AX5000_S_0104 :
STRUCT
	Position_loop_Kv_factor:UINT;
END_STRUCT
END_TYPE

// ---- POUs/IO/Drives/SoE/Ax5000ParamSTRUCTs/S/AX5000_S_0106.TcDUT
TYPE AX5000_S_0106 :
STRUCT
	Current_loop_proportional_gain_1:UINT;
END_STRUCT
END_TYPE

// ---- POUs/IO/Drives/SoE/Ax5000ParamSTRUCTs/S/AX5000_S_0111.TcDUT
TYPE AX5000_S_0111 :
STRUCT
	Motor_continouse_stall_current:UINT;
END_STRUCT
END_TYPE

// ---- POUs/IO/Drives/SoE/Ax5000ParamSTRUCTs/S/AX5000_S_0119.TcDUT
TYPE AX5000_S_0119 :
STRUCT
	Current_loop_proportional_gain2:UINT;
END_STRUCT
END_TYPE

// ---- POUs/IO/Drives/SoE/Ax5000ParamSTRUCTs/S/AX5000_S_0126.TcDUT
TYPE AX5000_S_0126 :
STRUCT
	Torque_threshold_Tx:UINT;
END_STRUCT
END_TYPE

// ---- POUs/IO/Drives/SoE/Ax5000ParamSTRUCTs/S/AX5000_S_0131.TcDUT
TYPE AX5000_S_0131 :
STRUCT
	Probe_value_1_negative_edge:DINT;
END_STRUCT
END_TYPE

// ---- POUs/IO/Drives/SoE/Ax5000ParamSTRUCTs/S/AX5000_S_0134.TcDUT
TYPE AX5000_S_0134 :
STRUCT
	Master_controll_word:UINT;
END_STRUCT
END_TYPE

// ---- POUs/IO/Drives/SoE/Ax5000ParamSTRUCTs/S/AX5000_S_0159.TcDUT
TYPE AX5000_S_0159 :
STRUCT
	Monitoring_window:UDINT;
END_STRUCT
END_TYPE

// ---- POUs/IO/Drives/SoE/Ax5000ParamSTRUCTs/S/AX5000_S_0160.TcDUT
TYPE AX5000_S_0160 :
STRUCT
	Acceleration_data_scaling_type:UINT;
END_STRUCT
END_TYPE

// ---- POUs/IO/Drives/SoE/Ax5000ParamSTRUCTs/S/AX5000_S_0161.TcDUT
TYPE AX5000_S_0161 :
STRUCT
	Acceleration_data_scaling_factor:UINT;
END_STRUCT
END_TYPE

// ---- POUs/IO/Drives/SoE/Ax5000ParamSTRUCTs/S/AX5000_S_0162.TcDUT
TYPE AX5000_S_0162 :
STRUCT
	Acceleration_data_scaling_exponent:UINT;
END_STRUCT
END_TYPE

// ---- POUs/IO/Drives/SoE/Ax5000ParamSTRUCTs/S/AX5000_S_0163.TcDUT
TYPE AX5000_S_0163 :
STRUCT
	Weight_counterbalance:INT;
END_STRUCT
END_TYPE

// ---- POUs/IO/Drives/SoE/Ax5000ParamSTRUCTs/S/AX5000_S_0179.TcDUT
TYPE AX5000_S_0179 :
STRUCT
	Probe_status:UINT;
END_STRUCT
END_TYPE

// ---- POUs/IO/Drives/SoE/Ax5000ParamSTRUCTs/S/AX5000_S_0185.TcDUT
TYPE AX5000_S_0185 :
STRUCT
	Length_of_the_configurabel_data_record_in_the_AT:UINT;
END_STRUCT
END_TYPE

// ---- POUs/IO/Drives/SoE/Ax5000ParamSTRUCTs/S/AX5000_S_0187.TcDUT
TYPE AX5000_S_0187 :
STRUCT
	Actual_lenght:UINT;
	Max_lenght:UINT;
	IDN_list_of_configurable_data_in_the_AT:ARRAY[0..67] OF UINT;
END_STRUCT
END_TYPE

// ---- POUs/IO/Drives/SoE/Ax5000ParamSTRUCTs/S/AX5000_S_0188.TcDUT
TYPE AX5000_S_0188 :
STRUCT
	Actual_lenght:UINT;
	Max_lenght:UINT;
	IDN_list_of_configurable_data_in_the_AT:ARRAY[0..13] OF UINT;
END_STRUCT
END_TYPE

// ---- POUs/IO/Drives/SoE/Ax5000ParamSTRUCTs/S/AX5000_S_0200.TcDUT
TYPE AX5000_S_0200 :
STRUCT
	Amplifier_warning_temperature:UINT;
END_STRUCT
END_TYPE

// ---- POUs/IO/Drives/SoE/Ax5000ParamSTRUCTs/S/AX5000_S_0216.TcDUT
TYPE AX5000_S_0216 :
STRUCT
	Switch_parameter:UINT;
END_STRUCT
END_TYPE

// ---- POUs/IO/Drives/SoE/Ax5000ParamSTRUCTs/S/AX5000_S_0217.TcDUT
TYPE AX5000_S_0217 :
STRUCT
	Parameter_set_preselection:UINT;
END_STRUCT
END_TYPE

// ---- POUs/IO/Drives/SoE/Ax5000ParamSTRUCTs/S/AX5000_S_0267.TcDUT
TYPE AX5000_S_0267 :
STRUCT
	Actual_lenght:UINT;
	Max_lenght:UINT;
	Password:STRING(29);
END_STRUCT
END_TYPE

// ---- POUs/IO/Drives/SoE/Ax5000ParamSTRUCTs/S/AX5000_S_0274.TcDUT
TYPE AX5000_S_0274 :
STRUCT
	Actual_lenght:UINT;
	Max_lenght:UINT;
	Received_drive_addresses:UINT;
END_STRUCT
END_TYPE

// ---- POUs/IO/Drives/SoE/Ax5000ParamSTRUCTs/S/AX5000_S_0372.TcDUT
TYPE AX5000_S_0372 :
STRUCT
	Drive_Halt_acceleration_bipolar:DINT;
END_STRUCT
END_TYPE

// ---- POUs/IO/Drives/SoE/Ax5000ParamSTRUCTs/S/AX5000_S_0375.TcDUT
TYPE AX5000_S_0375 :
STRUCT
	Actual_lenght:UINT;
	Max_lenght:UINT;
	Diagnostic_number_list:ARRAY[0..59] OF UINT;
END_STRUCT
END_TYPE

// ---- POUs/IO/Drives/SoE/Ax5000ParamSTRUCTs/S/AX5000_S_0380.TcDUT
TYPE AX5000_S_0380 :
STRUCT
	DC_bus_voltage:UINT;
END_STRUCT
END_TYPE

// ---- POUs/IO/Drives/SoE/Ax5000ParamSTRUCTs/S/AX5000_S_0383.TcDUT
TYPE AX5000_S_0383 :
STRUCT
	Motor_temperature:UINT;
END_STRUCT
END_TYPE

// ---- POUs/IO/Drives/SoE/Ax5000ParamSTRUCTs/S/AX5000_S_0429.TcDUT
TYPE AX5000_S_0429 :
STRUCT
	Emergancey_stop_decleration:UDINT;
END_STRUCT
END_TYPE

// ---- POUs/IO/Drives/SoE/Ax5000ParamSTRUCTs/S/AX5000_S_0435.TcDUT
TYPE AX5000_S_0435 :
STRUCT
	Operating_time_drive_control:UDINT;
END_STRUCT
END_TYPE

// ---- POUs/Logging/LogbookData.TcDUT
TYPE LogbookData :
STRUCT
	Timestamp												:	TIMESTRUCT;						//Stored timestamp for each message
	Msg														:	STRING(PARAM.LOGBOOK_MAX_MSG_STRING_LENGHT); //Stored message
{attribute 'displaymode':='binary'}	
	Options													:	WORD;							//Stored option for each message
END_STRUCT
END_TYPE

// ---- POUs/Motion/TF511x-KIN/03_DUTs/Positions/KIN_POSITIONS_MCS_DUT.TcDUT
TYPE KIN_POSITIONS_MCS_DUT EXTENDS VALUE_6D_DUT:
STRUCT
	Q1					: LREAL; //Auxiliary axis 1
	Q2					: LREAL; //Auxiliary axis 2 	
END_STRUCT
END_TYPE

// ---- POUs/Motion/TF511x-KIN/03_DUTs/Positions/U_KIN_POSITIONS.TcDUT
TYPE U_KIN_POSITIONS :  //Union datatype for kinematic positions in different identifier
UNION
	MCS							:	KIN_POSITIONS_MCS_DUT; //XYZ ABC Q1,Q2
	ACS							:	KIN_POSITIONS_ACS_DUT; //A1..A6,Q1,Q2
	Joints						:	ARRAY[1..8] OF LREAL; //Array 1..8
END_UNION
END_TYPE

// ---- POUs/Motion/VALUE_6D_DUT.TcDUT
TYPE VALUE_6D_DUT EXTENDS VALUE_3D_DUT:
STRUCT
	A					:		LREAL; //Rx
	B					:		LREAL; //Ry
	C					:		LREAL; //Rz	
END_STRUCT
END_TYPE

// ---- POUs/_Miscellaneous/U_32BIT_DATATYPE.TcDUT
TYPE U_32BIT_DATATYPE :  //Union datatype of 32 bit size datatypes 
UNION
	_REAL				: REAL;  
	{attribute 'displaymode':='hex'}	
	_DWORD				: DWORD;
	_DINT				: DINT;
	_UDINT				: UDINT;
	_TIME				: TIME;	
	_SINTS				: ARRAY[0..3] OF SINT; //Array 0..3 of BYTE
	{attribute 'displaymode':='hex'}	
	_BYTES				: ARRAY[0..3] OF BYTE; //Array 0..3 of BYTE
	{attribute 'displaymode':='hex'}	
	_WORDS				: ARRAY[0..1] OF WORD;	//Array 0..1 of WORD
	_INTS				: ARRAY[0..1] OF INT;	//Array 0..1 of INT
	_UINTS				: ARRAY[0..1] OF UINT;	//Array 0..1 of UINT
	
END_UNION
END_TYPE

// ---- POUs/_Miscellaneous/U_64BIT_DATATYPE.TcDUT
TYPE U_64BIT_DATATYPE : //Union datatype of 64 bit size datatypes 
UNION
//Native 64bit data types
	_LREAL													:	LREAL; 
	_LINT													:	LINT;
	_ULINT													:	ULINT;
	_LTIME													:	LTIME;
	{attribute 'displaymode':='hex'}                         	
	_LWORD													:	LWORD;	
	                    
//Alternative 64bit size variables as arrays of smaller datatypes                                     	
	_DINTs				 									:	ARRAY[0..1] OF DINT; //Array 0..1 of DINT
	_UDINTs													:	ARRAY[0..1] OF UDINT; //Array 0..1 of UDINT
	_INTs													: 	ARRAY[0..3] OF INT;	//Array 0..3 of INT
	_UINTs													: 	ARRAY[0..3] OF UINT;//Array 0..3 of UINT 
	_SINTs													: 	ARRAY[0..7] OF SINT;//Array 0..7 of SINT (signed 8bit)
	{attribute 'displaymode':='hex'}	                     	
	_BYTEs													:	ARRAY[0..7] OF BYTE; //Array 0..7 of BYTE
	{attribute 'displaymode':='hex'}	                     	
	_WORDs													:	ARRAY[0..3] OF WORD; //Array 0..3 of WORD
	{attribute 'displaymode':='hex'}	                     	
	_DWORDs													:	ARRAY[0..1] OF DWORD; //Array 0..1 of DWORD
END_UNION
END_TYPE

// ---- POUs/Statemodel/eSTATE.TcDUT
{attribute 'qualified_only'}
//Statemodel enum states 0 and 301-320
{attribute 'to_string'}
TYPE eSTATE :
(
	IDLE			:= 0,

	STARTUP			:= 301,
	ABORTING		:= 302,	
	ABORTED			:= 303,
	CLEARING		:= 304,

	STOPPING		:= 305,
	STOPPED			:= 306,
	RESETTING		:= 307,

	STARTING		:= 308,
	STARTED			:= 309,
	EXECUTE			:= 310,
	COMPLETING		:= 311,
	COMPLETE		:= 312,
	
	SUSPENDING		:= 313,
	SUSPENDED		:= 314,
	UNSUSPENDING	:= 315,
	HOLDING			:= 316,
	HELD			:= 317,
	UNHOLDING		:= 318
	);
END_TYPE

// ---- POUs/StringHelper/ExtendedString/T_EXT_STRING.TcDUT
TYPE T_EXT_STRING : STRING(PARAM.MAX_EXT_STRING_LENGTH); END_TYPE

// ---- POUs/StringHelper/ExtendedString/T_EXT_WSTRING.TcDUT
TYPE T_EXT_WSTRING : WSTRING(Param.MAX_EXT_STRING_LENGTH); END_TYPE

// ---- POUs/StringHelper/U_MAX_STRING.TcDUT
TYPE U_MAX_STRING :
UNION
	text				:	STRING(MAX_STRING_LENGTH);
	{attribute 'displaymode':='hex'}
	_BYTES				:	ARRAY[0..MAX_STRING_LENGTH] OF BYTE;	
END_UNION
END_TYPE

// ---- POUs/StringHelper/U_MAX_WSTRING.TcDUT
TYPE U_MAX_WSTRING :
UNION
	text				:	WSTRING(MAX_STRING_LENGTH);
	{attribute 'displaymode':='hex'}
	_BYTES				:	ARRAY[0..MAX_STRING_LENGTH] OF WORD;	
END_UNION
END_TYPE

// ---- GVLs/Gvl.TcGVL
VAR_GLOBAL
	{info <'Please check the disclaimer note vis function DisclaimerStatement (FUN) '>}
	
	CheckBoundsInfo												: 	CheckBoundsInfo; //Checkbounds result buffer 
	EventHandlingStatistic										:	EventHandlingStatisticInfo; //System information of eventlogger 
//	SOURCE_ID													:	SOURCE_ID; //Systemsource ids

	ALWAYS_TRUE										AT  %Q* 	:	BOOL := TRUE;
END_VAR
VAR_GLOBAL CONSTANT
	IBN															: 	BOOL := TRUE;	
END_VAR

// ---- GVLs/PARAM.TcGVL
{attribute 'qualified_only'}
VAR_GLOBAL CONSTANT
//Debug messages											
	ENABLE_DEBUG_MSG_DYNAMIC_MEM_ALLOCATION					:	BOOL := TRUE; //FBs who are allocating memory from the router memory pool via __NEW are writing a message into the ADS logger	

//Controller Tools
	SLIDING_AVERAGE_MAX_ENTRYS								:	INT := 1000;

//String helper
	MAX_EXT_STRING_LENGTH									:	UDINT := 1024; //Max string lenght for extended string FBs (ExtString,ExtWSTRING)	
	XWORD_TO_XXXSTR_EXT_SEPARATOR							:	STRING := '_';

//Data buffer settings
	RINGBUFFER_BYTE_SIMPLE_MAX_BUFFER						:	UDINT := 1024;	//Max index byte ringbuffer array
	RINGBUFFER_CHAR_SIMPLE_MAX_BUFFER						:	UDINT := 1024;	//Max index byte ringbuffer array for chars 	
	RINGBUFFER_LREAL_SIMPLE_MAX_BUFFER						:	UDINT := 10;	//Max index lreal ringbuffer array
	RINGBUFFER_REAL_SIMPLE_MAX_BUFFER						:	UDINT := 10;	//Max index real ringbuffer array
	
	FIFO_LREAL_SIMPEL_MAX_BUFFER							:	INT := 10;		//Max index lreal fifo array
	LIFO_LREAL_SIMPEL_MAX_BUFFER							:	INT := 10;		//Max index lreal lifo array	
	
//File handling 
	READ_DIR_SIMPLE_MAX_ENTRYS								:	INT(1..1000) := 50;	//Max list size of founded files in directory
	READ_DIR_SIMPLE_MAX_STRING_LEN							:	INT := 50;		//Maximum string lenght of files founded in directory
	
//Eventlogger  
	EVENT_HANDLING_CONFIG									:	EVENT_HANDLING_CONFIG  := (
																	GRP_CUSTOMISED_MAX_EVENT			:= 30,		
																	
																	EVENTLOG_READ_MSG_LEN_MIN			:= 0,
																	EVENTLOG_READ_MSG_LEN_MAX			:= 1024,
																	                                    
																	EVENTLOG_READ_MAX_EVENTS			:= 30,		
																	
																	ENABLE_DYNAMIC_EVENT_MSG_FORMAT		:= FALSE,
																	                                    
																	CLASS_NONE_QUIT_REQUIRED			:= FALSE,  	//Class id 0
																	CLASS_MAINTENANCE_QUIT_REQUIRED		:= TRUE,	//Class id 1	
																	CLASS_MESSAGE_QUIT_REQUIRED			:= FALSE,	//Class id 2
																	CLASS_HINT_QUIT_REQUIRED			:= FALSE,	//Class id 3
																	CLASS_STATEINFO_QUIT_REQUIRED		:= FALSE,	//Class id 4
																	CLASS_INSTRUCTION_QUIT_REQUIRED		:= FALSE,	//Class id 5
																	CLASS_WARNING_QUIT_REQUIRED			:= TRUE,	//Class id 6
																	CLASS_ALARM_QUIT_REQUIRED			:= TRUE,	//Class id 7
																	CLASS_PARAMERROR_QUIT_REQUIRED		:= TRUE,	//Class id 8
																	                                    
																	CLASS_NONE_PRIORITY					:= 3,
																	CLASS_MAINTENANCE_PRIORITY			:= 2,
																	CLASS_MESSAGE_PRIORITY				:= 3,
																	CLASS_HINT_PRIORITY					:= 3,
																	CLASS_STATEINFO_PRIORITY			:= 3,
																	CLASS_INSTRUCTION_PRIORITY			:= 3,
																	CLASS_WARNING_PRIORITY				:= 2,   
																	CLASS_ALARM_PRIORITY				:= 1,		
																	CLASS_PARAMERROR_PRIORITY			:= 1);	
		
//Logbook settings 
	LOGBOOK_MAX_DATA										:	INT(1..1000) := 50; //no of messages stored in the PLC - logbook
	LOGBOOK_MAX_MSG_STRING_LENGHT							:	UDINT := 255; //Max sring lenght of logbook message
	LOGBOOK_PUPLISHER_MAX_SUB								:	INT := 5;
	LOGBOOK_SUB_WRT_FILE_LINE_END_SIGN						:	STRING(6) := '$n'; //line end sign
	LOGBOOK_SUB_WRT_FILE_DELAY_FILE_CLOSE					:	TIME := T#5S; //Delay close logbook file and release handle 
	LOGBOOK_SUB_MAX_EVENT_HANDLING							:	UINT(1..100) := 10; //no of EventHandling instances to display logbook entrys
	LOGBOOK_SUB_SEND_MAIL_STR_LINE_END_SIGN					:	STRING(6) := '$r$n'; //line end sign
	
			
//Statemodel control settings
	STATEMODEL_CTRL_MAX_SLAVE								:	INT(1..100) := 8; //no of possible subs for each state model master instance
	
//IO-Fieldbus Master
	ETHERCAT_MASTER_DEV_IO_MAX_FRAMES						:	INT := 4;
	ETHERCAT_DIAG_MAX_SLAVES								:	UINT := 100;
	
	PROFIBUS_MASTER_DEV_IO_MAX_SLAVES						:	INT := 10;
	PROFINET_DEVICE_DEV_IO_MAX_BOX 							:	INT := 1;
	PROFINET_CONTROLLER_DEV_IO_MAX_BOX 						:	INT := 10;

//IO
	ETHERCAT_SLAVE_DEV_FW_UPDATER_MAX_DEV					:	INT := 10;	
	
//Safety 
	SAFETY_PLC_TERM_DIAG_MAX_FB								:	INT := 30;
	SAFETY_IO_TERM_DIAG_MAX									:	INT := 10;
	SAFETY_LOGIC_IO_TERM_DIAG_MAX_MODULE					:	int := 8;
	
//Quicksort settings
	QUICKSORT_MAX_STRING_LENGTH								:	INT := 256;
	QUICKSORT_MAX_WSTRING_LENGTH							:	INT := 256;
	
//Modbus 
	MODBUS_MAX_SLAVE_JOB									:	INT := 10;
	MODBUS_MAX_SLAVES_OF_MASTER								:	INT := 10;
	
//Device Com array limits
	DEVICE_COM_MIN_CACHE									:	INT := 0;	//UNION type DeviceCom Cache MIN  
	DEVICE_COM_MAX_CACHE									:	INT := 1024;//UNION type DeviceCom Cache MAX  

END_VAR

// ---- Version/Global_Version.TcGVL
{attribute 'TcGenerated'}
{attribute 'no-analysis'}
{attribute 'linkalways'}
// This function has been automatically generated from the project information.
VAR_GLOBAL CONSTANT
	{attribute 'const_non_replaced'}
	stLibVersion_EngineeringToolbox : ST_LibVersion := (iMajor := 3, iMinor := 1, iBuild := 2, iRevision := 3, nFlags := 1, sVersion := '3.1.2.3');
END_VAR

// ---- POUs/IO/Drives/I_AxDriveBase.TcIO
INTERFACE I_AxDriveBase EXTENDS __SYSTEM.IQueryInterface

PROPERTY PUBLIC rAxDrive : REFERENCE TO AxDriveBase
GET
END_GET
END_PROPERTY

END_INTERFACE

// ---- POUs/IO/_EcSlaveInfoDataIO/I_EcSlaveInfoData.TcIO
INTERFACE I_EcSlaveInfoData EXTENDS __SYSTEM.IQueryInterface

PROPERTY PUBLIC rInfoData : reference to EcSlaveInfoData
GET
END_GET
END_PROPERTY

END_INTERFACE

// ---- POUs/IO/_ItfActuators/I_ActuatorFwdRev.TcIO
INTERFACE I_ActuatorFwdRev EXTENDS I_ActuatorBase

{attribute 'monitoring' := 'call'}
PROPERTY public forwardStarted : BOOL
GET
END_GET
END_PROPERTY

{attribute 'monitoring' := 'call'}
PROPERTY public reverseStarted : BOOL
GET
END_GET
END_PROPERTY

METHOD public startForward : BOOL
VAR_INPUT
END_VAR
END_METHOD

METHOD public startReverse : BOOL
VAR_INPUT
END_VAR
END_METHOD

END_INTERFACE

// ---- POUs/IO/_ItfActuators/I_ActuatorFwdBwd.TcIO
INTERFACE I_ActuatorFwdBwd EXTENDS I_ActuatorBase

{attribute 'monitoring' := 'call'}
PROPERTY public backwardStarted : BOOL
GET
END_GET
END_PROPERTY

{attribute 'monitoring' := 'call'}
PROPERTY public forwardStarted : BOOL
GET
END_GET
END_PROPERTY

METHOD public startBackward : BOOL
VAR_INPUT
END_VAR
END_METHOD

METHOD public startForward : BOOL
VAR_INPUT
END_VAR
END_METHOD

END_INTERFACE

// ---- POUs/IO/_ItfActuators/I_ActuatorLeftRight.TcIO
INTERFACE I_ActuatorLeftRight EXTENDS I_ActuatorBase

{attribute 'monitoring' := 'call'}
PROPERTY public leftOk : BOOL
GET
END_GET
END_PROPERTY

{attribute 'monitoring' := 'call'}
PROPERTY public rightOk : BOOL
GET
END_GET
END_PROPERTY

METHOD public toTheLeft : BOOL
VAR_INPUT
END_VAR
END_METHOD

METHOD public toTheRight : BOOL
VAR_INPUT
END_VAR
END_METHOD

END_INTERFACE

// ---- POUs/Statemodel/UnitTemplate/I_Statemodel_Unit.TcIO
INTERFACE I_Statemodel_Unit Extends __System.IQueryInterface

{attribute 'monitoring' := 'call'}
PROPERTY public rUnit : REFERENCE TO Statemodel
GET
END_GET
END_PROPERTY

END_INTERFACE

// ---- POUs/Motion/TF50xx-NC/00_Base/I_AxNcBase.TcIO
INTERFACE I_AxNcBase EXTENDS __SYSTEM.IQueryInterface

METHOD PUBLIC noAction : BOOL //Return value = TRUE if busy of home and motion 
VAR_INPUT
END_VAR
END_METHOD

{attribute 'monitoring' := 'call'}
PROPERTY rAdmin : REFERENCE TO AxAdmin
GET
END_GET
END_PROPERTY

{attribute 'monitoring' := 'call'}
PROPERTY rAxisRef : REFERENCE TO AXIS_REF
GET
END_GET
END_PROPERTY

{attribute 'monitoring' := 'call'}
PROPERTY rErrHdl : REFERENCE to ERROR_HDL
GET
END_GET
SET
END_SET
END_PROPERTY

METHOD reset : Bool
VAR_INPUT
END_VAR
END_METHOD

{attribute 'monitoring' := 'call'}
PROPERTY rHome : REFERENCE TO AxHoming
GET
END_GET
END_PROPERTY

{attribute 'monitoring' := 'call'}
PROPERTY rPara : REFERENCE TO AxPara
GET
END_GET
END_PROPERTY

END_INTERFACE

// ---- Version/disclaimerStatement.TcPOU
// .. Disclaimer:: This function contains statements about the use of this library 
{attribute 'no-analysis'}
{attribute 'no_check'}
FUNCTION disclaimerStatement : WSTRING(1500)
VAR_INPUT
END_VAR
VAR
END_VAR

DisclaimerStatement := 
	"This disclaimer contains statements about the use of this library.

		-The use of this version of the library is free of charge 
		-It is incumbent on the customer to check and decide whether the library and provided function is suitable for use his particular application
		-This library is provided 'AS IS' and neither a part of TwinCAT3 nor directly supported by Beckhoff Automation
		-The use of the Library is at the Customer's own risk
		-There is no warranty given that the library and source code, which is made available with this library is complete or accurate
		-In no event will the author or Beckhoff Automation be liable for any claims, damages or other liability for errors and/or omissions arising from the use of the library
		-There is no right to expect maintenance, support, enhancements or modifications of the library as well as for updates or compatibility to updates of the library or TwinCAT3 if released
		
	For feedback or questions please contact the Beckhoff Industry Management for Electronics Manufacturing, D.Schlingmann@Beckhoff.com
	
	© Beckhoff Automation GmbH & Co. KG,
	The reproduction, distribution and utilisation of this library or parts of it as well as the communication of its content to others without express authorisation is prohibited held liable for the payment of damages.
	
	All rights reserved in the event of the grant of a patent, utility model or design.";

END_FUNCTION

// ---- POUs/BoundsCheck/CheckBoundsInfo.TcPOU
//CheckBoundsInfo creates a an message entry in the TwinCAT logger 
//and provides information about the number of bounds errors as well signal variables if an error occured.
//Example of TwinCAT logger message: 	'Array index too low! Lower: 1 Upper: 10 Index: 11'
//
//please copy code example for CheckBounds as shown at this code section below into your "CheckBounds (FUN)"
{attribute 'no_check'}
FUNCTION_BLOCK CheckBoundsInfo
VAR_INPUT
	Interlock												:	BOOL; //TestAndSet interlock for multicore use
END_VAR                 									
VAR_OUTPUT              									
	LogMsg													:	T_MAXSTRING; 	//Last ADS log message
	CountUpper												:	UDINT := 0; 	//Counter of CheckBounds errors if index is greater the the upper limit 
	CountLower												:	UDINT := 0;		//Counter of CheckBounds errors if index is smaller the the lower limit 
	ErrorUpper												:	BOOL;			//Error upper limit occured - see LogMsg for further information
	ErrorLower												:	BOOL;			//Error lower limit occured - see LogMsg for further information
END_VAR                 									
VAR                     	
	MEM														:	ARRAY[1..3] OF DINT;
END_VAR

(* 
//Code template for implicit check function of "CheckBounds (FUN)"
IF  index < lower 
THEN
	(* Return right index *)
	CheckBounds 											:= lower;	

	IF TestAndSet(ET.CheckBoundsInfo.Interlock)
	THEN
		ET.CheckBoundsInfo.SetErrorLower(index,lower,upper);
		ET.CheckBoundsInfo.Interlock						:= FALSE;
	END_IF

ELSIF index > upper 
THEN
	(* Return right index *)
	CheckBounds 											:= upper;
	
	IF TestAndSet(ET.CheckBoundsInfo.Interlock)
	THEN
		ET.CheckBoundsInfo.SetErrorUpper(index,lower,upper);
		ET.CheckBoundsInfo.Interlock						:= FALSE;
	END_IF
	
ELSE  
	CheckBounds 											:= index;
END_IF
*)

METHOD PUBLIC reset : BOOL //Return value = TRUE if execution finished
VAR_INPUT
END_VAR
IF 	ErrorUpper OR ErrorLower
THEN
	CountUpper 												:= CountLower := 0;
	ErrorUpper												:= FALSE;
	ErrorLower												:= FALSE;
	MEMSET(ADR(MEM),0,SIZEOF(MEM));
END_IF
reset														:= TRUE;
END_METHOD

METHOD PUBLIC setErrorLower : booL //called by implicit function CheckBounds
VAR_INPUT
	index, lower, upper: DINT;
END_VAR
LogMsg														:=CONCAT('Array index too low! Index:',DINT_TO_STRING(index));
LogMsg														:=CONCAT(LogMsg,', Lower:');
LogMsg														:=CONCAT(LogMsg,DINT_TO_STRING(Lower));
LogMsg														:=CONCAT(LogMsg,', Upper:');
LogMsg														:=CONCAT(LogMsg,DINT_TO_STRING(Upper));
                                                        	
CountLower 													:= CountLower +1;                                                   	
ErrorLower													:= TRUE;
                                                        	
// write daten into eventlogger                         	
IF	lower <> MEM[1]                                     	
	OR Upper <> MEM[2]                                  	
	OR Index <> MEM[3]                                  	
THEN                                                    	
	ADSLOGDINT(	ADSLOG_MSGTYPE_ERROR OR ADSLOG_MSGTYPE_LOG,
				LogMsg,
				0);
END_IF

// store errors in memorybuffer
MEM[1] 														:= lower;
MEM[2] 														:= Upper;
MEM[3] 														:= index;

setErrorLower												:= TRUE;
END_METHOD

METHOD PUBLIC setErrorUpper :booL//called by implicit function CheckBounds
VAR_INPUT
	index, lower, upper: DINT;
END_VAR
LogMsg															:=CONCAT('Array index too high! Index:',DINT_TO_STRING(index));
LogMsg															:=CONCAT(LogMsg,', Lower:');
LogMsg															:=CONCAT(LogMsg,DINT_TO_STRING(Lower));
LogMsg															:=CONCAT(LogMsg,', Upper:');
LogMsg															:=CONCAT(LogMsg,DINT_TO_STRING(Upper));

CountUpper 														:= CountUpper +1;
ErrorUpper														:= TRUE;

// write daten into eventlogger
IF lower <> MEM[1]
	OR Upper <> MEM[2]
	OR Index <> MEM[3]
THEN
	ADSLOGDINT(	ADSLOG_MSGTYPE_ERROR OR ADSLOG_MSGTYPE_LOG,
					LogMsg,
					0);
END_IF

// store errors in memorybuffer
MEM[1] 															:= lower;
MEM[2] 															:= Upper;
MEM[3] 															:= index;

setErrorUpper													:= TRUE;
END_METHOD

END_FUNCTION_BLOCK

// ---- POUs/BoundsCheck/checkBounds.TcPOU
//Implicit function for checking array bounds - called by system
//This check bounds implementation includes "CheckBoundsInfo (FB)", which is already an instance object of this library and can be found at ET.<Gvl>.CheckBoundsInfo.
//CheckBoundsInfo creates a an entry in the TwinCAT logger and provides information about the number of errors and signal variables if an error occures.
//Example of TwinCAT logger message: 	'Array index too low! Lower: 1 Upper: 10 Index: 11'
//
//please copy code example as shown after END_VAR as a command.
FUNCTION checkBounds : DINT
VAR_INPUT
	Index, Lower, Upper: DINT;
END_VAR

IF  index < lower 
THEN
	(* Return right index *)
	CheckBounds 											:= lower;	

	//
	IF TestAndSet(ET.CheckBoundsInfo.Interlock)
	THEN
		ET.CheckBoundsInfo.SetErrorLower(index,lower,upper);
		ET.CheckBoundsInfo.Interlock						:= FALSE;
	END_IF

ELSIF index > upper 
THEN
	(* Return right index *)
	CheckBounds 											:= upper;
	
	IF TestAndSet(ET.CheckBoundsInfo.Interlock)
	THEN
		ET.CheckBoundsInfo.SetErrorUpper(index,lower,upper);
		ET.CheckBoundsInfo.Interlock						:= FALSE;
	END_IF
	
ELSE  
	CheckBounds 											:= index;
END_IF

END_FUNCTION

// ---- POUs/EventLogger/TriggerEvents/EventHandlingStatisticInfo.TcPOU
{attribute 'no_check'}
//Collection with count and class types of active events 
FUNCTION_BLOCK EventHandlingStatisticInfo
VAR_OUTPUT CONSTANT
	MIN_CLASS												: 	UINT := TCEVENTCLASS_NONE;
	MAX_CLASS												: 	UINT := TCEVENTCLASS_PARAMERROR;
	MIN_PRIORITY											: 	INT := 0;
	MAX_PRIORITY											: 	INT := 7;
END_VAR
VAR_INPUT
	ClassInfo												:	ARRAY[MIN_CLASS..MAX_CLASS] OF INT; (* No of active messages in each class
																										TCEVENTCLASS_NONE			:=0
																										TCEVENTCLASS_MAINTENANCE	:=1	
																										TCEVENTCLASS_MESSAGE		:=2
																										TCEVENTCLASS_HINT			:=3	
																										TCEVENTCLASS_STATEINFO		:=4	
																										TCEVENTCLASS_INSTRUCTION	:=5	
																										TCEVENTCLASS_WARNING		:=6	
																										TCEVENTCLASS_ALARM			:=7	
																										TCEVENTCLASS_PARAMERROR		:=8 *)
	PriorityInfo											:	ARRAY[MIN_PRIORITY..MAX_PRIORITY] OF INT; //No of active messages per priority - see Param.EVENT_HANDLING_CONFIG
	NoOfQuitRequiredEvents									:	INT;
	NoOfActiveEvents										:	INT;
END_VAR
VAR_OUTPUT
END_VAR
VAR
	TaskInterlockCountIn									:	BOOL;
	TaskInterlockCountOut									:	BOOL;
END_VAR

;

PROPERTY PUBLIC classAlarmActive : BOOL
GET
classAlarmActive													:= ClassInfo[TCEVENTCLASS_ALARM] <> 0;
END_GET
END_PROPERTY

PROPERTY PUBLIC classHintActive : BOOL
GET
classHintActive													:= ClassInfo[TCEVENTCLASS_HINT] <> 0;
END_GET
END_PROPERTY

PROPERTY PUBLIC classInstructionActive : BOOL
GET
classInstructionActive													:= ClassInfo[TCEVENTCLASS_INSTRUCTION] <> 0;
END_GET
END_PROPERTY

PROPERTY PUBLIC classMaintenanceActive : BOOL
GET
classMaintenanceActive													:= ClassInfo[TCEVENTCLASS_MAINTENANCE] <> 0;
END_GET
END_PROPERTY

PROPERTY PUBLIC classMessageActive : BOOL
GET
classMessageActive													:= ClassInfo[TCEVENTCLASS_MESSAGE] <> 0;
END_GET
END_PROPERTY

PROPERTY PUBLIC classNoneActive : BOOL
GET
ClassNoneActive													:= ClassInfo[TCEVENTCLASS_NONE] <> 0;
END_GET
END_PROPERTY

PROPERTY PUBLIC classParamErrorActive : BOOL
GET
ClassParamErrorActive													:= ClassInfo[TCEVENTCLASS_PARAMERROR] <> 0;
END_GET
END_PROPERTY

PROPERTY PUBLIC classStateinfoActive : BOOL
GET
ClassStateinfoActive													:= ClassInfo[TCEVENTCLASS_STATEINFO] <> 0;
END_GET
END_PROPERTY

PROPERTY PUBLIC classWarningActive : BOOL
GET
ClassWarningActive													:= ClassInfo[TCEVENTCLASS_WARNING] <> 0;
END_GET
END_PROPERTY

METHOD PUBLIC clear : BOOL //Return value = TRUE if execution finished 
VAR_INPUT
END_VAR
	MEMSET(ADR(ClassInfo),0,SIZEOF(ClassInfo));
	MEMSET(ADR(PriorityInfo),0,SIZEOF(PriorityInfo));
	NoOfQuitRequiredEvents									:= 0;	
	NoOfActiveEvents										:= 0;
	Clear													:= TRUE;
END_METHOD

{attribute 'hide'}
METHOD PUBLIC countIn : BOOL //Return value = TRUE if execution finished 
VAR_IN_OUT
	Status													:	DWORD; (*	.0 - .8 = event of <class id> is active / .15 confirm required / .16 = Level 0 , .17 = Level 1 , .18 = Level 2, ..........
																			TCEVENTCLASS_NONE			:=0,	(* No class *)
																			TCEVENTCLASS_MAINTENANCE	:=1,	(* Maintenance hint *)
																			TCEVENTCLASS_MESSAGE		:=2,	(* Message *)
																			TCEVENTCLASS_HINT			:=3,	(* Hint *)
																			TCEVENTCLASS_STATEINFO		:=4,	(* State information *)
																			TCEVENTCLASS_INSTRUCTION	:=5,	(* Instruction *)
																			TCEVENTCLASS_WARNING		:=6,	(* Warning *)
																			TCEVENTCLASS_ALARM			:=7,	(* Alarm *)
																			TCEVENTCLASS_PARAMERROR		:=8		(* Parameter error *)  *)
END_VAR
IF TestAndSet(TaskInterlockCountIn)
THEN
	IF Status.0 THEN ClassInfo[TCEVENTCLASS_NONE] 				:= ClassInfo[TCEVENTCLASS_NONE] + 1; 									
	ELSIF Status.1 THEN ClassInfo[TCEVENTCLASS_MAINTENANCE] 	:= ClassInfo[TCEVENTCLASS_MAINTENANCE] + 1; 
	ELSIF Status.2 THEN ClassInfo[TCEVENTCLASS_MESSAGE] 		:= ClassInfo[TCEVENTCLASS_MESSAGE] + 1; 	
	ELSIF Status.3 THEN ClassInfo[TCEVENTCLASS_HINT] 			:= ClassInfo[TCEVENTCLASS_HINT] + 1; 		
	ELSIF Status.4 THEN ClassInfo[TCEVENTCLASS_STATEINFO] 		:= ClassInfo[TCEVENTCLASS_STATEINFO] + 1; 	
	ELSIF Status.5 THEN ClassInfo[TCEVENTCLASS_INSTRUCTION] 	:= ClassInfo[TCEVENTCLASS_INSTRUCTION] + 1; 
	ELSIF Status.6 THEN ClassInfo[TCEVENTCLASS_WARNING] 		:= ClassInfo[TCEVENTCLASS_WARNING] + 1; 	
	ELSIF Status.7 THEN ClassInfo[TCEVENTCLASS_ALARM] 			:= ClassInfo[TCEVENTCLASS_ALARM] + 1; 		
	ELSIF Status.8 THEN ClassInfo[TCEVENTCLASS_PARAMERROR] 		:= ClassInfo[TCEVENTCLASS_PARAMERROR] + 1; 	
	END_IF
	
	IF Status.15 THEN NoOfQuitRequiredEvents 					:= NoOfQuitRequiredEvents + 1; END_IF
	
	IF status.16 THEN PriorityInfo[0]							:= PriorityInfo[0] + 1;						
	ELSIF status.17 THEN PriorityInfo[1]						:= PriorityInfo[1] + 1	;						
	ELSIF status.18 THEN PriorityInfo[2]						:= PriorityInfo[2] + 1;						
	ELSIF status.19 THEN PriorityInfo[3]						:= PriorityInfo[3] + 1;						
	ELSIF status.20 THEN PriorityInfo[4]						:= PriorityInfo[4] + 1;						
	ELSIF status.21 THEN PriorityInfo[5]						:= PriorityInfo[5] + 1;						
	ELSIF status.22 THEN PriorityInfo[6]						:= PriorityInfo[6] + 1;						
	ELSIF status.23 THEN PriorityInfo[7]						:= PriorityInfo[7] + 1	;						
	END_IF
	
	//set active flag	
	NoOfActiveEvents											:= NoOfActiveEvents + 1;
	
	status.31 													:= TRUE; 
	CountIn														:= TRUE;
	TaskInterlockCountIn										:= FALSE;
END_IF
END_METHOD

// {attribute 'hide'}
METHOD PUBLIC countOut : BOOL //Return value = TRUE if execution finished 
VAR_IN_OUT
	Status													:	DWORD; (*	.0 - .8 = event of <class id> is active / .15 confirm required / .16 = Level 0 , .17 = Level 1 , .18 = Level 2, ..........
																			TCEVENTCLASS_NONE			:=0,	(* No class *)
																			TCEVENTCLASS_MAINTENANCE	:=1,	(* Maintenance hint *)
																			TCEVENTCLASS_MESSAGE		:=2,	(* Message *)
																			TCEVENTCLASS_HINT			:=3,	(* Hint *)
																			TCEVENTCLASS_STATEINFO		:=4,	(* State information *)
																			TCEVENTCLASS_INSTRUCTION	:=5,	(* Instruction *)
																			TCEVENTCLASS_WARNING		:=6,	(* Warning *)
																			TCEVENTCLASS_ALARM			:=7,	(* Alarm *)
																			TCEVENTCLASS_PARAMERROR		:=8		(* Parameter error *)  *)
END_VAR
IF TestAndSet(TaskInterlockCountOut)
THEN
	IF Status.0 THEN ClassInfo[TCEVENTCLASS_NONE] 				:= MAX(0,ClassInfo[TCEVENTCLASS_NONE] - 1); 		
	ELSIF Status.1 THEN ClassInfo[TCEVENTCLASS_MAINTENANCE] 	:= MAX(0,ClassInfo[TCEVENTCLASS_MAINTENANCE] - 1);	
	ELSIF Status.2 THEN ClassInfo[TCEVENTCLASS_MESSAGE] 		:= MAX(0,ClassInfo[TCEVENTCLASS_MESSAGE] - 1); 		
	ELSIF Status.3 THEN ClassInfo[TCEVENTCLASS_HINT] 			:= MAX(0,ClassInfo[TCEVENTCLASS_HINT] - 1); 		
	ELSIF Status.4 THEN ClassInfo[TCEVENTCLASS_STATEINFO] 		:= MAX(0,ClassInfo[TCEVENTCLASS_STATEINFO] - 1); 	
	ELSIF Status.5 THEN ClassInfo[TCEVENTCLASS_INSTRUCTION] 	:= MAX(0,ClassInfo[TCEVENTCLASS_INSTRUCTION] - 1);	
	ELSIF Status.6 THEN ClassInfo[TCEVENTCLASS_WARNING] 		:= MAX(0,ClassInfo[TCEVENTCLASS_WARNING] - 1); 	
	ELSIF Status.7 THEN ClassInfo[TCEVENTCLASS_ALARM] 			:= MAX(0,ClassInfo[TCEVENTCLASS_ALARM] - 1); 		
	ELSIF Status.8 THEN ClassInfo[TCEVENTCLASS_PARAMERROR] 		:= MAX(0,ClassInfo[TCEVENTCLASS_PARAMERROR] - 1); 	
	END_IF
																	  
	IF Status.15 THEN NoOfQuitRequiredEvents 					:=  MAX(0,NoOfQuitRequiredEvents - 1); 	
	END_IF
																	   
	IF status.16 THEN PriorityInfo[0]							:=  MAX(0,PriorityInfo[0] - 1);						
	ELSIF status.17 THEN PriorityInfo[1]						:=  MAX(0,PriorityInfo[1] - 1);						
	ELSIF status.18 THEN PriorityInfo[2]						:=  MAX(0,PriorityInfo[2] - 1);						
	ELSIF status.19 THEN PriorityInfo[3]						:=  MAX(0,PriorityInfo[3] - 1);						
	ELSIF status.20 THEN PriorityInfo[4]						:=  MAX(0,PriorityInfo[4] - 1);						
	ELSIF status.21 THEN PriorityInfo[5]						:=  MAX(0,PriorityInfo[5] - 1);						
	ELSIF status.22 THEN PriorityInfo[6]						:=  MAX(0,PriorityInfo[6] - 1);						
	ELSIF status.23 THEN PriorityInfo[7]						:=  MAX(0,PriorityInfo[7] - 1);						
	END_IF
	
	NoOfActiveEvents											:= MAX(0,NoOfActiveEvents - 1);
	status.31													:= FALSE; //Active flag reset
	CountOut													:= TRUE;
	TaskInterlockCountOut										:= FALSE;
END_IF
END_METHOD

METHOD INTERNAL initEvent : DWORD //Return status 
VAR_IN_OUT
	SetClass								:	E_TcEventClass;
	EventConfig								:	TcEvent;
END_VAR
		(* Event Config *)
		InitEvent											:= 0;
		IF SetClass = TC2_SYSTEM.TCEVENTCLASS_NONE 				
		THEN	
			EventConfig.Class								:= SetClass;
			EventConfig.bQuitRequired						:= PARAM.EVENT_HANDLING_CONFIG.CLASS_NONE_QUIT_REQUIRED;
			InitEvent.15									:= PARAM.EVENT_HANDLING_CONFIG.CLASS_NONE_QUIT_REQUIRED;
			EventConfig.Prio								:= PARAM.EVENT_HANDLING_CONFIG.CLASS_NONE_PRIORITY;
			InitEvent										:= SETBIT32(InitEvent,TO_SINT(PARAM.EVENT_HANDLING_CONFIG.CLASS_NONE_PRIORITY) + 16);	
			InitEvent.0										:= TRUE;													
			
		ELSIF SetClass = TC2_SYSTEM.TCEVENTCLASS_MAINTENANCE 
		THEN
			EventConfig.Class								:= SetClass;
			EventConfig.bQuitRequired						:= PARAM.EVENT_HANDLING_CONFIG.CLASS_MAINTENANCE_QUIT_REQUIRED;
			InitEvent.15									:= PARAM.EVENT_HANDLING_CONFIG.CLASS_MAINTENANCE_QUIT_REQUIRED;
			EventConfig.Prio								:= PARAM.EVENT_HANDLING_CONFIG.CLASS_MAINTENANCE_PRIORITY;
			InitEvent										:= SETBIT32(InitEvent,TO_SINT(PARAM.EVENT_HANDLING_CONFIG.CLASS_MAINTENANCE_PRIORITY) + 16);
			InitEvent.1										:= TRUE;
		ELSIF SetClass = TC2_SYSTEM.TCEVENTCLASS_MESSAGE 		
		THEN
			EventConfig.Class								:= SetClass;
			EventConfig.bQuitRequired						:= PARAM.EVENT_HANDLING_CONFIG.CLASS_MESSAGE_QUIT_REQUIRED;
			InitEvent.15									:= PARAM.EVENT_HANDLING_CONFIG.CLASS_MESSAGE_QUIT_REQUIRED;
			EventConfig.Prio								:= PARAM.EVENT_HANDLING_CONFIG.CLASS_MESSAGE_PRIORITY;
			InitEvent										:= SETBIT32(InitEvent,TO_SINT(PARAM.EVENT_HANDLING_CONFIG.CLASS_MESSAGE_PRIORITY) + 16);
			InitEvent.2										:= TRUE;
		ELSIF SetClass = TC2_SYSTEM.TCEVENTCLASS_HINT 			
		THEN
			EventConfig.Class								:= SetClass;
			EventConfig.bQuitRequired						:= PARAM.EVENT_HANDLING_CONFIG.CLASS_HINT_QUIT_REQUIRED;
			InitEvent.15									:= PARAM.EVENT_HANDLING_CONFIG.CLASS_HINT_QUIT_REQUIRED;
			EventConfig.Prio								:= PARAM.EVENT_HANDLING_CONFIG.CLASS_HINT_PRIORITY;
			InitEvent										:= SETBIT32(InitEvent,TO_SINT(PARAM.EVENT_HANDLING_CONFIG.CLASS_HINT_PRIORITY) + 16);
			InitEvent.3										:= TRUE;
		ELSIF SetClass = TC2_SYSTEM.TCEVENTCLASS_STATEINFO 	
		THEN
			EventConfig.Class								:= SetClass;
			EventConfig.bQuitRequired						:= PARAM.EVENT_HANDLING_CONFIG.CLASS_STATEINFO_QUIT_REQUIRED;
			InitEvent.15									:= PARAM.EVENT_HANDLING_CONFIG.CLASS_STATEINFO_QUIT_REQUIRED;
			EventConfig.Prio								:= PARAM.EVENT_HANDLING_CONFIG.CLASS_STATEINFO_PRIORITY;
			InitEvent										:= SETBIT32(InitEvent,TO_SINT(PARAM.EVENT_HANDLING_CONFIG.CLASS_STATEINFO_PRIORITY) + 16);
			InitEvent.4										:= TRUE;
		ELSIF SetClass = TC2_SYSTEM.TCEVENTCLASS_INSTRUCTION 
		THEN
			EventConfig.Class								:= SetClass;
			EventConfig.bQuitRequired						:= PARAM.EVENT_HANDLING_CONFIG.CLASS_INSTRUCTION_QUIT_REQUIRED;
			InitEvent.15									:= PARAM.EVENT_HANDLING_CONFIG.CLASS_INSTRUCTION_QUIT_REQUIRED;
			EventConfig.Prio								:= PARAM.EVENT_HANDLING_CONFIG.CLASS_INSTRUCTION_PRIORITY;
			InitEvent										:= SETBIT32(InitEvent,TO_SINT(PARAM.EVENT_HANDLING_CONFIG.CLASS_INSTRUCTION_PRIORITY) + 16);
			InitEvent.5										:= TRUE;
		ELSIF SetClass = TC2_SYSTEM.TCEVENTCLASS_WARNING 		
		THEN
			EventConfig.Class								:= SetClass;
			EventConfig.bQuitRequired						:= PARAM.EVENT_HANDLING_CONFIG.CLASS_WARNING_QUIT_REQUIRED;
			InitEvent.15									:= PARAM.EVENT_HANDLING_CONFIG.CLASS_WARNING_QUIT_REQUIRED;
			EventConfig.Prio								:= PARAM.EVENT_HANDLING_CONFIG.CLASS_WARNING_PRIORITY;
			InitEvent										:= SETBIT32(InitEvent,TO_SINT(PARAM.EVENT_HANDLING_CONFIG.CLASS_WARNING_PRIORITY) + 16);
			InitEvent.6										:= TRUE;
		ELSIF SetClass = TC2_SYSTEM.TCEVENTCLASS_ALARM 		
		THEN
			EventConfig.Class								:= SetClass;
			EventConfig.bQuitRequired						:= PARAM.EVENT_HANDLING_CONFIG.CLASS_ALARM_QUIT_REQUIRED;
			InitEvent.15									:= PARAM.EVENT_HANDLING_CONFIG.CLASS_ALARM_QUIT_REQUIRED;
			EventConfig.Prio								:= PARAM.EVENT_HANDLING_CONFIG.CLASS_ALARM_PRIORITY;
			InitEvent										:= SETBIT32(InitEvent,TO_SINT(PARAM.EVENT_HANDLING_CONFIG.CLASS_ALARM_PRIORITY) + 16);
			InitEvent.7										:= TRUE;
		ELSIF SetClass = TC2_SYSTEM.TCEVENTCLASS_PARAMERROR 	
		THEN
			EventConfig.Class								:= SetClass;
			EventConfig.bQuitRequired						:= PARAM.EVENT_HANDLING_CONFIG.CLASS_PARAMERROR_QUIT_REQUIRED;
			InitEvent.15									:= PARAM.EVENT_HANDLING_CONFIG.CLASS_PARAMERROR_QUIT_REQUIRED;
			EventConfig.Prio								:= PARAM.EVENT_HANDLING_CONFIG.CLASS_PARAMERROR_PRIORITY;
			InitEvent										:= SETBIT32(InitEvent,TO_SINT(PARAM.EVENT_HANDLING_CONFIG.CLASS_PARAMERROR_PRIORITY) + 16);
			InitEvent.8										:= TRUE;
		ELSE 
			EventConfig.Class								:= SetClass;
			EventConfig.bQuitRequired						:= PARAM.EVENT_HANDLING_CONFIG.CLASS_ALARM_QUIT_REQUIRED;
			InitEvent.15									:= PARAM.EVENT_HANDLING_CONFIG.CLASS_ALARM_QUIT_REQUIRED;
			EventConfig.Prio								:= PARAM.EVENT_HANDLING_CONFIG.CLASS_ALARM_PRIORITY;
			InitEvent										:= SETBIT32(InitEvent,TO_SINT(PARAM.EVENT_HANDLING_CONFIG.CLASS_ALARM_PRIORITY) + 16);
			InitEvent.7										:= TRUE;
		END_IF
END_METHOD

METHOD PUBLIC isClassActive : BOOL  //Return value = TRUE if EventClass is currently active
VAR_INPUT
	TcEventClass											:	E_TcEventClass;
END_VAR
IF TcEventClass < MIN_CLASS OR TcEventClass > MAX_CLASS
THEN
	IsClassActive											:= TRUE;
ELSE
	IsClassActive											:= ClassInfo[TcEventClass] <> 0;
END_IF
END_METHOD

PROPERTY PUBLIC isConfirmReqActive : BOOL
GET
isConfirmReqActive											:= NoOfQuitRequiredEvents <> 0;
END_GET
END_PROPERTY

METHOD PUBLIC isPriorityActive : BOOL //Return value = TRUE if priority is active
VAR_INPUT
	IN														:	INT;
END_VAR
IF IN < MIN_PRIORITY OR IN > MAX_PRIORITY
THEN
	IsPriorityActive										:= TRUE;
ELSE
	IsPriorityActive										:= PriorityInfo[In] <> 0;
END_IF
END_METHOD

END_FUNCTION_BLOCK

// ---- POUs/EventLogger/TriggerEvents/EventHandling.TcPOU
{attribute 'no_check'}
//ADSLOGEVENT wrapper for a convenient and pre configured use - see Beckhoff documentation for more information about AdsEventLogger
//See Param constanst to configure whether the TcEventClass need to be acknowledged (confirmation required) 
FUNCTION_BLOCK EventHandling
VAR_INPUT
	Flag													:	BOOL := FALSE; //Fire event 
	ConfirmTrig												:	BOOL := FALSE; //Ack event
	MsgId													:	UINT := 0; //Event number
	SourceId												: 	UDINT:= 0; //Event source number
	eClass													:	E_TcEventClass := TCEVENTCLASS_ALARM; (*	TC2_SYSTEM.TCEVENTCLASS_NONE		
																											TC2_SYSTEM.TCEVENTCLASS_MAINTENANCE
																											TC2_SYSTEM.TCEVENTCLASS_MESSAGE		
																											TC2_SYSTEM.TCEVENTCLASS_HINT		
																											TC2_SYSTEM.TCEVENTCLASS_STATEINFO	
																											TC2_SYSTEM.TCEVENTCLASS_INSTRUCTION	
																											TC2_SYSTEM.TCEVENTCLASS_WARNING		
																											TC2_SYSTEM.TCEVENTCLASS_ALARM		
																											TC2_SYSTEM.TCEVENTCLASS_PARAMERROR	*)

	Text1													:	STRING(20) := ''; //Short info text with lenght 20 chars 
	Text2													:	STRING(40) := ''; //Long info text with lenght 40 chars
	pText3													:	POINTER TO STRING := 0; //Pointer to extended info text 
END_VAR
VAR_OUTPUT
{attribute 'displaymode':='hex'}
	State													:	UDINT ; (*	TCEVENTSTATE_INVALID  	: WORD := 16#0000; 		
																			TCEVENTSTATE_SIGNALED  	: WORD := 16#0001; 		- The event is signaled 
																			TCEVENTSTATE_RESET  	: WORD := 16#0002; 		- The event is gone 
																			TCEVENTSTATE_CONFIRMED  : WORD := 16#0010 (16); - The event is confirmed 
																			TCEVENTSTATE_RESETCON  	: WORD := 16#0012 (18); - The event is gone AND confirmed *)
{attribute 'displaymode':='binary'}
	Status													:	DWORD; (*	.0 - .8 = event <class id>  / .15 confirm required / .16 = Level 0 , .17 = Level 1 , .18 = Level 2, .......... / .31 active
																			TCEVENTCLASS_NONE			:=0,
																			TCEVENTCLASS_MAINTENANCE	:=1,
																			TCEVENTCLASS_MESSAGE		:=2,
																			TCEVENTCLASS_HINT			:=3,
																			TCEVENTCLASS_STATEINFO		:=4, 
																			TCEVENTCLASS_INSTRUCTION	:=5,
																			TCEVENTCLASS_WARNING		:=6,
																			TCEVENTCLASS_ALARM			:=7,
																			TCEVENTCLASS_PARAMERROR		:=8	 *)
END_VAR
VAR
	format													:	STRING(6) := '%s%s%s';
	pPara													:	ARRAY[1..3] OF POINTER TO BYTE;
	TmpString												:	STRING(1) := '';
	AdsEvent												:	ADSLOGEVENT :=(
																	NETID				:= '',
																	PORT				:= AMSPORT_EVENTLOG,
																	TMOUT 				:= DEFAULT_ADS_TIMEOUT,
																	EventDataLength		:= 0,	
																	EventConfigData 	:= (
																		Class 				:= TCEVENTCLASS_ALARM,
																		Prio 				:= TCEVENTPRIO_IMPLICIT,
																		ProgId 				:= 'TcEventFormatter.TcXmlFormatter',
																		Flags 				:= TCEVENTFLAG_LOG OR TCEVENTFLAG_SRCID, // 16#0140 (* T *),
																		StreamType 			:= TCEVENTSTREAM_SIMPLE (* TCEVENTSTREAM_NORMAL *),
																		bQuitRequired 		:= TRUE));
END_VAR

(* EventHandling including textinfos which are send to the eventlogger  	v4.3	*)
(* specific eventclasses have to be quit, see Param.EventConfig...					*)
(************************************************************************************)

(* sequence *************************************************************)
	IF Status.31 //Message active
	THEN (* work EventLogger *)
		AdsEvent(
			NETID			:= ,(* see declaration *)
			PORT			:= ,(* see declaration *)
			Event			:= NOT AdsEvent.FbCleanup AND(Flag OR AdsEvent.EventState = TCEVENTSTATE_INVALID AND NOT AdsEvent.Quit), (* Set Event until state <> invalid *)
			EventQuit		:= AdsEvent.EventState <> TCEVENTSTATE_INVALID
								AND AdsEvent.EventConfigData.bQuitRequired
								AND NOT AdsEvent.Eventstate.4 //confirmed
								AND NOT AdsEvent.Quit
								AND(
								ConfirmTrig
								OR AdsEvent.EventQuit), (* quit send *)
			EventConfigData	:= ,(* see declaration *)
			EventDataAddress:= ADR(pPara),
			EventDataLength	:= ,(* see declaration *)
			FbCleanup		:= NOT AdsEvent.FbCleanup AND(AdsEvent.Err OR AdsEvent.EventState = TCEVENTSTATE_RESETCON),
			TMOUT			:= ,(* see declaration *)
			EventState		=> ,
			Err				=> ,
			ErrId			=> ,
			Quit			=> );
			
		IF AdsEvent.Event 
			AND AdsEvent.EventState = TCEVENTSTATE_INVALID
		THEN
			State 											:= SEL(Flag, TCEVENTSTATE_RESET, TCEVENTSTATE_SIGNALED);
		ELSIF AdsEvent.Quit
			AND AdsEvent.EventState = TCEVENTSTATE_INVALID
			AND AdsEvent.EventQuit
			OR 
			AdsEvent.FbCleanup		
		THEN
			State 											:= TCEVENTSTATE_RESETCON;
		ELSIF(AdsEvent.Err OR NOT AdsEvent.Event AND AdsEvent.EventState = TCEVENTSTATE_INVALID)
			AND_THEN Gvl.EventHandlingStatistic.CountOut(Status)
		THEN
			State											:= TCEVENTSTATE_INVALID;
		ELSE
			State											:= MAX(State, AdsEvent.EventState);
		END_IF
			
	ELSIF Flag AND SourceId > 0 
	THEN (* fire event *)
		IF PARAM.EVENT_HANDLING_CONFIG.ENABLE_DYNAMIC_EVENT_MSG_FORMAT
		THEN
			IF pText3 <> 0 AND_THEN pText3^[0] > 0
			THEN 
				format 										:= '%s%s%s'; 
			ELSIF Text2[0] > 0 
			THEN 
				format 										:= '%s%s';
			ELSIF Text1[0] > 0 
			THEN 												
				format 										:= '%s';
			ELSE
				format 										:= '';
			END_IF
		END_IF
							 
		AdsEvent.EventConfigData.DataFormatStrAddress		:= ADR(format);
		AdsEvent.EventConfigData.Id 						:= UINT_TO_UDINT(MsgID);
		AdsEvent.EventConfigData.SourceId 					:= SourceId;
		Status												:= Gvl.EventHandlingStatistic.InitEvent(SetClass := eClass, EventConfig := AdsEvent.EventConfigData);		

		(* Data *)
		pPara[1] 											:= ADR(Text1);
		pPara[2] 											:= ADR(Text2);
		pPara[3] 											:= SEL(pText3 <> 0,ADR(TmpString) ,pText3);
	
		IF AdsEvent.Err AND NOT AdsEvent.FbCleanup
		THEN
			AdsEvent(
				Event			:= FALSE,
				EventQuit 		:= FALSE,
				EventDataAddress:= ADR(pPara),
				FbCleanup		:= TRUE,
				EventState		=> );
				
		ELSE (* Fire Event *)
			AdsEvent( 	
				Event			:= FALSE,
				EventQuit 		:= FALSE, 
				FbCleanup 		:= FALSE, 
				EventDataAddress:= ADR(pPara));
						
			AdsEvent( 	Event 	:= TRUE);
			IF NOT AdsEvent.Err AND_THEN Gvl.EventHandlingStatistic.CountIn(Status) //Add event to statistic and continue if added successfully
			THEN			
				State 										:= TCEVENTSTATE_SIGNALED;
			END_IF
						
		END_IF
	END_IF

(**********************************************************************************)

END_FUNCTION_BLOCK

